// TwinCAT 3 PLC project CAP_TESTER
// ProgramVersion: 3.1.4023.0
// libraries:
//   Tc2_ControllerToolbox, * (Beckhoff Automation GmbH)
//   Tc2_Standard, * (Beckhoff Automation GmbH)
//   Tc2_System, * (Beckhoff Automation GmbH)
//   Tc2_Utilities, * (Beckhoff Automation GmbH)
//   Tc3_Module, * (Beckhoff Automation GmbH)
// project tree:
//   DUTs/ BIT2.TcDUT, ST_AnalogCHSelection.TcDUT
//   GVLs/ GVL.TcGVL, HMI_DB.TcGVL, LV.TcGVL, VoltMonitor_DB.TcGVL
//   / PlcTask.TcTTO
//   POUs/ ADC_10V.TcPOU, ADC_5V.TcPOU, ALIAS.TcPOU, ANALOGConversion.TcPOU, Automated_Capacitor_Test_ST.TcPOU, CounterUP.TcPOU, handleFAULT.TcPOU, handlesensorlimitFAULTS.TcPOU, handlesoftEXCEPTION.TcPOU, HMI.TcPOU, LV_ALIAS.TcPOU, MAIN.TcPOU, Norm_x.TcPOU, PRG_FB_CTRL_PWM_OUT.TcPOU, VoltMonitor.TcPOU
//   POUs/Functions/AnalogIN-ScaleOffset/ AI2temp.TcPOU, AI1temp.TcPOU, AI3temp.TcPOU, AI4temp.TcPOU
//   POUs/Functions/AnalogIN-ScaleOffset/Voltage Calibration/ AI5volt.TcPOU
//   POUs/Functions/AnalogOut-ScaleOffset/ volt_TO_AO1_802L50kV.TcPOU
//   POUs/Functions/ estimatedchargeTIME_802L.TcPOU, HV_Monitor.TcPOU, instantexpectedcapVOLT_802L.TcPOU, Heartbeat.TcPOU, Norm_x_UINT.TcPOU, tempSAFE.TcPOU
// real-time tasks:
//   TASK PlcTask: cycle T#10ms, priority 20, ADS port 350
// I/O:
//   DEVICE Device 1 (EtherCAT), AmsNetId 172.25.226.104.2.1
//     Term 1 (EK1200) [EK1200-5000 EtherCAT Power supply (2A E-Bus)]
//       Term 2 (EL1008) [EL1008 8Ch. Dig. Input 24V, 3ms]
//       Term 3 (EL1008) [EL1008 8Ch. Dig. Input 24V, 3ms]
//       Term 4 (EL2008) [EL2008 8Ch. Dig. Output 24V, 0.5A]
//       Term 5 (EL2008) [EL2008 8Ch. Dig. Output 24V, 0.5A]
//       Term 6 (EL3064) [EL3064 4Ch. Ana. Input 0-10V]
//       Term 7 (EL3064) [EL3064 4Ch. Ana. Input 0-10V]
//       Term 8 (EL3064) [EL3064 4Ch. Ana. Input 0-10V]
//       Term 9 (EL4132) [EL4132 2Ch. Ana. Output +/-10V, 16bit]
//       Term 10 (EL9011) [EL9011 End Terminal]
//   DEVICE Device 3 (RT-Ethernet Protocol) (disabled), AmsNetId 172.25.226.104.4.1
//   DEVICE Device 2 (NOV-DP-RAM) (disabled)
//   DEVICE Device 6 (EtherCAT), AmsNetId 5.97.49.116.7.1
//     Box 11 (170357) [170357]
// variable links:
//   CAP_TESTER/CAP_TESTER Instance <-> Device 1 (EtherCAT)/Term 1 (EK1200)/Term 2 (EL1008)
//     PlcTask Inputs/GVL.PLC_DI{1..8} <-> Channel {1..8}/Input  (8 links)
//   CAP_TESTER/CAP_TESTER Instance <-> Device 1 (EtherCAT)/Term 1 (EK1200)/Term 3 (EL1008)
//     PlcTask Inputs/GVL.PLC_DI{9..16} <-> Channel {1..8}/Input  (8 links)
//   CAP_TESTER/CAP_TESTER Instance <-> Device 1 (EtherCAT)/Term 1 (EK1200)/Term 4 (EL2008)
//     PlcTask Outputs/GVL.PLC_DO{1..8} <-> Channel {1..8}/Output  (8 links)
//   CAP_TESTER/CAP_TESTER Instance <-> Device 1 (EtherCAT)/Term 1 (EK1200)/Term 5 (EL2008)
//     PlcTask Outputs/GVL.PLC_DO{9..16} <-> Channel {1..8}/Output  (8 links)
//   CAP_TESTER/CAP_TESTER Instance <-> Device 1 (EtherCAT)/Term 1 (EK1200)/Term 6 (EL3064)
//     PlcTask Inputs/GVL.PLC_AI{1..4} <-> AI Standard Channel {1..4}/Value  (4 links)
//     PlcTask Inputs/GVL.PLC_AI{1..4}_LIM1 <-> AI Standard Channel {1..4}/Status  (4 links)
//   CAP_TESTER/CAP_TESTER Instance <-> Device 1 (EtherCAT)/Term 1 (EK1200)/Term 7 (EL3064)
//     PlcTask Inputs/GVL.PLC_AI{5..8} <-> AI Standard Channel {1..4}/Value  (4 links)
//     PlcTask Inputs/GVL.PLC_AI{5..8}_LIM1 <-> AI Standard Channel {1..4}/Status  (4 links)
//   CAP_TESTER/CAP_TESTER Instance <-> Device 1 (EtherCAT)/Term 1 (EK1200)/Term 8 (EL3064)
//     PlcTask Inputs/GVL.PLC_AI{9..12} <-> AI Standard Channel {1..4}/Value  (4 links)
//     PlcTask Inputs/GVL.PLC_AI{9..12}_LIM1 <-> AI Standard Channel {1..4}/Status  (4 links)
//   CAP_TESTER/CAP_TESTER Instance <-> Device 1 (EtherCAT)/Term 1 (EK1200)/Term 9 (EL4132)
//     PlcTask Outputs/GVL.PLC_AO1 <-> Channel 1/Output
//     PlcTask Outputs/GVL.PLC_AO2 <-> Channel 2/Output
//   CAP_TESTER/CAP_TESTER Instance <-> Device 6 (EtherCAT)/Box 11 (170357)
//     PlcTask Inputs/GVL.B170357_CapRaw[{0..24}] <-> HV Cap process data mapping/Cap {0..24} Raw  (25 links)

CONFIGURATION CAP_TESTER
    RESOURCE PLC ON TwinCAT3
        TASK PlcTask(INTERVAL := T#10ms, PRIORITY := 20);
        PROGRAM MAIN WITH PlcTask : MAIN;
    END_RESOURCE
END_CONFIGURATION

// ---- DUTs/BIT2.TcDUT
(* STRUCT typedef for EL3XXX AI BIT2 limit *)
TYPE BIT2 :
STRUCT
	BIT_0: BIT;		// < or =< is BIT0 true 
	BIT_1: BIT;		// > or => is BIT1 true
END_STRUCT
END_TYPE

// ---- DUTs/ST_AnalogCHSelection.TcDUT
TYPE ST_AnalogCHSelection :
STRUCT
	b0 : BIT;
	b1 : BIT;
	b2 : BIT;
	b3 : BIT;
END_STRUCT
END_TYPE

// ---- GVLs/GVL.TcGVL
{attribute 'qualified_only'}
VAR_GLOBAL

 //Alwas True & False
 AlwaysTrue : BOOL := TRUE;
 AlwaysFalse : BOOL := FALSE;
 
(* PLC Physical IO *)
	// Digital IO
	buttonSTOP : BOOL;		// Unused
	mechINTERLOCK : BOOL;
	softdump : BOOL := FALSE; 
	softdump_contact : BOOL;   // soft dump relay feedback. Normally Closed - ctrl box dump feedback is the soft dump feedback, in here ctrlbox dump feedback is not used
	chargeCOIL : BOOL := FALSE;
	chargeCOIL_contact : BOOL; // charge coil relay feedback. Normally Open
	shotCOIL : BOOL := FALSE;
	shotCOILrdy : BOOL;
	testFAULTlight : BOOL;
	testRUNlight : BOOL;
	scopetrigger : BOOL;
	charging_alarm :BOOL;
	sparkdetect :BOOL;
	FireDetected :BOOL;  //Newly added for Fire Detection Test
	chrg_to_fire_trig :BOOL := FALSE; //debug signal for Firedetect system
	FruitStandDumpingON : BOOL := FALSE;
	
	(* For HVPS Controller IO *)
	psuVmonitor : INT;		// PLC in to V monitor, is psu V measurement. AI
	psuVCTRL : INT;		// PLC out to remote voltage, is psu V control. AO
	selectREMOTE : BOOL := FALSE;		// PLC out to remote/ local select, is psu ON/ OFF control.
	psuInhibit : BOOL := TRUE;		// PLC out to inhibit, inhibits psu.
	psuInhibit_contact : BOOL;		// No PCB with available signal thus unused.
	psuONOFF : BOOL;		// PLC in to High Voltage Monitor, is psu ON/ OFF status.
	EOCstatus : BOOL;		// PLC in to EOC, is psu End of Charge
	psuINTERLOCK : BOOL;		// PLC in
	psusumFAULT : BOOL;		// PLC in
	psuMaxOutput : UINT;  //Maximum output setting on a Charger Power supply  (12kV or 50kV) * added oct 12, 2022 GL
	
	sparkCharger_ON : BOOL;  // added output to turn on spark charger sept 21, 2022 GL
	sparkCharger_SP_Enable : BOOL; // added setpoint enable to spark charger sept 21, 2022 GL
	
	(* AI TEMP/ VOLT *)
	rawTEMPcap1 : INT; // Cap1 
		TEMPcap1 : INT;
	rawTEMPdump : INT; // Soft Dump
		TEMPdump : INT;
	rawTEMPload : INT; // Load 
		TEMPload : INT;
	rawTEMPambient : INT; // Ambient 
		TEMPambient : INT;
	rawVcap1 : INT;	// Cap1 Voltage
		Vcap1 : INT;
		changeAI5 :BOOL := FALSE;
	raw_HV_monitor : INT;
		HV_monitor :INT;
		
		Vcap2 : INT;  //Cap1 Voltage with 0-10V for testing oct, 27, 2022
		Vcap2_norm : REAL;
		Vcap2_REAL : REAL;
		
	raw_Spark_gap_voltage :INT;  //AI8 - added Oct 5, 2022 - GL
		Spark_gap_voltage :INT;
		Spark_gap_voltage_norm : REAL;
		Spark_gap_voltage_REAL : REAL;
	raw_VoltageMonitor : INT;
(* PLC Internal *)
	appRUN : BOOL;
	

	(* Manual HMI Controls *)
	HMIhold : BOOL;
	HMIcharge : BOOL;
	HMIdump : BOOL;
	HMIshoot : BOOL;
	HMIready : BOOL;
	
(* FAULTS *)
	chargeFAULT : BOOL := FALSE;
	dischargeFAULT : BOOL := FALSE;
	holdFAULT : BOOL := FALSE;
	cap1tempFAULT : BOOL := FALSE;
	ambienttempFAULT : BOOL := FALSE;
	loadtempFAULT : BOOL := FALSE;  // ADDED OCT 14, 2022 GL
	psuFAULT : BOOL := FALSE;
	ctrlsysFAULT : BOOL := FALSE;		// Relates to FB sys
		softdumpFB_FAULT : BOOL := FALSE;
		chargeFB_FAULT : BOOL := FALSE;
		HVpsuFB_FAULT : BOOL := FALSE;
	softexceptionFAULT : BOOL := FALSE;
	test_interval_fault : BOOL := FALSE;
	PreFire_Fault : BOOL := FALSE;

(*DEBUG*)
	ctrl_box_charge_feedback : BOOL;  //relay contact ??
	ctrl_box_dump_feedback : BOOL;	//relay contact ??
(* Start PLC ALIAS *)
		// Digital In
	PLC_DI1 AT %I* : BOOL;
	PLC_DI2 AT %I* : BOOL;
	PLC_DI3 AT %I* : BOOL;
	PLC_DI4 AT %I* : BOOL;
	PLC_DI5 AT %I* : BOOL;
	PLC_DI6 AT %I* : BOOL;
	PLC_DI7 AT %I* : BOOL;
	PLC_DI8 AT %I* : BOOL;
	PLC_DI9 AT %I* : BOOL;
	PLC_DI10 AT %I* : BOOL;
	PLC_DI11 AT %I* : BOOL;
	PLC_DI12 AT %I* : BOOL;
	PLC_DI13 AT %I* : BOOL;
	PLC_DI14 AT %I* : BOOL;
	PLC_DI15 AT %I* : BOOL;
	PLC_DI16 AT %I* : BOOL;
		// Digital Out
	PLC_DO1 AT %Q* : BOOL;
	PLC_DO2 AT %Q* : BOOL;
	PLC_DO3 AT %Q* : BOOL;
	PLC_DO4 AT %Q* : BOOL;
	PLC_DO5 AT %Q* : BOOL;
	PLC_DO6 AT %Q* : BOOL;
	PLC_DO7 AT %Q* : BOOL;
	PLC_DO8 AT %Q* : BOOL;
	PLC_DO9 AT %Q* : BOOL;
	PLC_DO10 AT %Q* : BOOL;
	PLC_DO11 AT %Q* : BOOL;
	PLC_DO12 AT %Q* : BOOL; //Voltage Monitor b0
	PLC_DO13 AT %Q* : BOOL; //Voltage Monitor b1
	PLC_DO14 AT %Q* : BOOL; //Voltage Monitor b2
	PLC_DO15 AT %Q* : BOOL; //Voltage Monitor b3
	PLC_DO16 AT %Q* : BOOL; //spare
		// Analog In
	PLC_AI1 AT %I* : INT;
	PLC_AI2 AT %I* : INT;
	PLC_AI3 AT %I* : INT;
	PLC_AI4 AT %I* : INT;
	PLC_AI5 AT %I* : INT;
	PLC_AI6 AT %I* : INT;
	PLC_AI7 AT %I* : INT;
	PLC_AI8 AT %I* : INT;
	PLC_AI9 AT %I* : INT;
	PLC_AI10 AT %I* : INT;
	PLC_AI11 AT %I* : INT;
	PLC_AI12 AT %I* : INT;
			// Analog Satus Limit WORD Bits 2/3 is Limit 1..... BIT.0 is WORD.2 and BIT.1 is WORD.3
			PLC_AI1_LIM1 AT %I*: WORD;
			PLC_AI2_LIM1 AT %I*: WORD;
			PLC_AI3_LIM1 AT %I*: WORD;
			PLC_AI4_LIM1 AT %I*: WORD;
			PLC_AI5_LIM1 AT %I*: WORD;
			PLC_AI6_LIM1 AT %I*: WORD;
			PLC_AI7_LIM1 AT %I*: WORD;
			PLC_AI8_LIM1 AT %I*: WORD;
			PLC_AI9_LIM1 AT %I*: WORD;
			PLC_AI10_LIM1 AT %I*: WORD;
			PLC_AI11_LIM1 AT %I*: WORD;
			PLC_AI12_LIM1 AT %I*: WORD;
		// Analog Out
	PLC_AO1 AT %Q* : INT;
	PLC_AO2 AT %Q* : INT;
	
	// PLC IO Status
	PLC_EL1008_1 AT %I* : UINT;
	PLC_EL1008_2 AT %I* : UINT;
	PLC_EL2008_1 AT %I* : UINT;
	PLC_EL2008_2 AT %I* : UINT;
	PLC_EL3064_1 AT %I* : UINT;
	PLC_EL3064_2 AT %I* : UINT;
	PLC_EL3064_3 AT %I* : UINT;
	PLC_EL4132_1 AT %I* : UINT;
	
	// EtherCAT Module
	DevCtrl AT %Q* : UINT;
	
	//customed board 170357
	(*B170357_CapRaw0 AT %I* : UINT;
	B170357_CapRaw1 AT %I* : UINT;
	B170357_CapRaw2 AT %I* : UINT;
	B170357_CapRaw3 AT %I* : UINT;
	B170357_CapRaw4 AT %I* : UINT;
	B170357_CapRaw5 AT %I* : UINT;
	B170357_CapRaw6 AT %I* : UINT;
	B170357_CapRaw7 AT %I* : UINT;
	B170357_CapRaw8 AT %I* : UINT;
	B170357_CapRaw9 AT %I* : UINT;
	B170357_CapRaw10 AT %I* : UINT;
	B170357_CapRaw11 AT %I* : UINT;
	B170357_CapRaw12 AT %I* : UINT;
	B170357_CapRaw13 AT %I* : UINT;
	B170357_CapRaw14 AT %I* : UINT;
	B170357_CapRaw15 AT %I* : UINT;
	B170357_CapRaw16 AT %I* : UINT;
	B170357_CapRaw17 AT %I* : UINT;
	B170357_CapRaw18 AT %I* : UINT;
	B170357_CapRaw19 AT %I* : UINT;
	B170357_CapRaw20 AT %I* : UINT;
	B170357_CapRaw21 AT %I* : UINT;
	B170357_CapRaw22 AT %I* : UINT;
	B170357_CapRaw23 AT %I* : UINT;
	B170357_CapRaw24 AT %I* : UINT;*)
	
	B170357_CapRaw AT %I* : ARRAY[0..24] OF UINT;
	B170357_BatLevel AT %I* : BOOL;
	B170357_Heartbeat AT %I* : BOOL;
	

END_VAR

VAR_GLOBAL PERSISTENT
	(* HMI IO *)
	hmiSTOP : BOOL; // In (Into PLC from LabView)
	hmiSTART : BOOL;	// In
	HOA : BOOL;	// In
	
	voltage_held_by_PSU :BOOL;
	isnotSCRhvswitch : BOOL;	// If HV switch has feedback. SCR has ready feedback signal.
	psu50kV_OutputSelected : BOOL; 
	Cap_ratedVoltage : UINT; // unit is in V
	targetVolt_exceed_CapRating_FAULT : BOOL;
	expectedvoltage : INT;
	psuTargetinvolt_echo : DINT;
	
	clearFAULT : BOOL;	// In
	
	testintervalsecs : INT; 	// In
	overall_cycle_time : INT;
	circuitcapacitanceuF : REAL;	// In
	cap1THRESHOLDcel : INT;	// In
	softdumpTHRESHOLDcel : INT := 95; // IN, added oct 14, 2022 GL
	loadTHRESHOLDcel : INT := 95;  // IN, added oct 14, 2022 GL
	ambientTHRESHOLDcel : INT := 95;  // IN, added oct 14, 2022 GL
	allTemperatureInRange : BOOL; //OUT, added oct 14, 2022 GL
	
	targetPSUVOLT : DINT;	// In 
	psuVOLTrating : DINT;	// In
	psuPOWERpeak : DINT;	// In
	chargeTIME : REAL;	// Out. Is estimated charge time of cap
	chargeTIMEmanual : REAL;	// In
	holdTIMEsec : REAL; // IN 
		holdTIMEtime : TIME;
	testNUM: INT;
	testNUMmax : INT;	// In
	testNUMexceed: BOOL;  //CHANGED FROM INT TO BOOL - JUNE 20, 2022
	resettestNUM : BOOL;	// In
	
	(* Current Control *)
	control_current : BOOL;
	duty_cycle : REAL;
	
	InstrumentationFault : BOOL := FALSE;
	noFaultDetected: BOOL := TRUE;
END_VAR

// ---- GVLs/HMI_DB.TcGVL
{attribute 'qualified_only'}
VAR_GLOBAL
	Fault: WORD; 
	
	Charging			: BOOL := FALSE;
	Dumping				: BOOL := FALSE;
	ActivateChargePB 	: BOOL := FALSE;
	ActivateDumpPB 		: BOOL := FALSE;
	
END_VAR

// ---- GVLs/LV.TcGVL
{attribute 'qualified_only'}
// variables to be used with LabVIEW
VAR_GLOBAL
	
aBools : ARRAY[1..20] OF BOOL;
aInts : ARRAY[1..10] OF INT;

END_VAR

// ---- GVLs/VoltMonitor_DB.TcGVL
{attribute 'qualified_only'}
VAR_GLOBAL
	Heartbeat : BOOL;
	BateryOn  : BOOL;
	Channel	: USINT; //ST_AnalogCHSelection;
	VoltageReading_raw : ARRAY[0..24] OF INT;
	VoltageReading_norm : ARRAY[0..24] OF REAL;
	VoltageReading	: ARRAY[0..15] OF REAL;
	LoadMaxRatedV	: REAL := 13800; //-2k TO 35kV
	LoadMinRatedV	: REAL := -1450; //Jake's lab result
	
	CapRaw : ARRAY[0..24] OF UINT;
	CapRawBIT : UINT;
	CapRaw_DummySnap : ARRAY[0..24] OF UINT;
	CapRaw_Str: STRING;
	BatteryLevel : BOOL;
	
	//cunter for missing packets
	missedCTU : CTU;
	//ONS	: R_TRIG;
	missingCNT : WORD :=0;
	
	Time1		: TON;
	Time1_ET	: TIME;
	packetsPerMin : REAL;
	//missedCTU : CTU;
	ONS	: R_TRIG;
	//missingCNT : WORD;
	missingCNT_REAL : REAL;
END_VAR

// ---- POUs/MAIN.TcPOU
PROGRAM MAIN

ALIAS();
LV_ALIAS();
ANALOGconversion();
handleFAULT();
handlesensorlimitFAULTS();
handlesoftEXCEPTION();
Automated_Capacitor_Test_ST();	
HMI();
HV_Monitor();
VoltMonitor();
//HMI Refresh clock
Heartbeat();
// runningLIGHTS();

END_PROGRAM

// ---- POUs/ALIAS.TcPOU
PROGRAM ALIAS
VAR
END_VAR

(* ALIAS Map 
Can be used for wiring and variable linking. ! Remember to SETUP and link AI1-4 LIMIT1 Bits !
Disclaimers: 
Digital IO PCB input Ch3/4 are inverted - No light in, 24V. Wired to PLC_DO6/7
Look at specifcations document for mapping.
*)
	// Digital Input
	GVL.mechINTERLOCK 			:= GVL.PLC_DI1 ;	// Normally Low when not interlock
	GVL.softdump_contact 		:= GVL.PLC_DI2 ;		// NL when no FB. Goes high when the relay is engaged and is not soft dumping. NO 
	GVL.psuONOFF 				:= GVL.PLC_DI3 ;	// To PSU High Voltage Monitor - Normally HIGH when HV OFF/ sig
	GVL.psusumFAULT 			:= GVL.PLC_DI4 ;	// To PSU Sum Fault - NH when no fault/ sig
	//GVL.psuINTERLOCK 			:= GVL.PLC_DI5 ;	// To PSU Interlock. Unknown if NH or NL
	GVL.ctrl_box_dump_feedback 	:= GVL.PLC_DI5;		// this variable is not used, softdump_contact is used instead and it is coming from the ctrlbox dump fb
	GVL.EOCStatus 				:= GVL.PLC_DI6 ;		// End of charge - NH when not EOC
	GVL.sparkdetect 			:= GVL.PLC_DI7 ;		// DI Extra1 - Mech TEST STOP sw - Normally LOW. Not used.
	GVL.chargeCOIL_contact 		:= GVL.PLC_DI8 ;	// NL
	GVL.shotCOILrdy 			:= GVL.PLC_DI9 ;		// NL
	GVL.FireDetected 			:= GVL.PLC_DI10 ;   // for Fire Detection
	GVL.FruitStandDumpingON		:= GVL.PLC_DI13;
	VoltMonitor_DB.Heartbeat 	:= GVL.B170357_Heartbeat;//:= GVL.PLC_DI11 ;   // Voltage Monitor Heartbeat
	VoltMonitor_DB.BateryOn		:= GVL.B170357_BatLevel;//:= GVL.PLC_DI12 ;
	VoltMonitor_DB.CapRaw[0]	:= GVL.B170357_CapRaw[0];
	VoltMonitor_DB.CapRaw[1]	:= GVL.B170357_CapRaw[1];
	VoltMonitor_DB.CapRaw[2]	:= GVL.B170357_CapRaw[2];
	VoltMonitor_DB.CapRaw[3]	:= GVL.B170357_CapRaw[3];
	VoltMonitor_DB.CapRaw[4]	:= GVL.B170357_CapRaw[4];
	VoltMonitor_DB.CapRaw[5]	:= GVL.B170357_CapRaw[5];
	VoltMonitor_DB.CapRaw[6]	:= GVL.B170357_CapRaw[6];
	VoltMonitor_DB.CapRaw[7]	:= GVL.B170357_CapRaw[7];
	VoltMonitor_DB.CapRaw[8]	:= GVL.B170357_CapRaw[8];
	VoltMonitor_DB.CapRaw[9]	:= GVL.B170357_CapRaw[9];
	VoltMonitor_DB.CapRaw[10]	:= GVL.B170357_CapRaw[10];
	VoltMonitor_DB.CapRaw[11]	:= GVL.B170357_CapRaw[11];
	VoltMonitor_DB.CapRaw[12]	:= GVL.B170357_CapRaw[12];
	VoltMonitor_DB.CapRaw[13]	:= GVL.B170357_CapRaw[13];
	VoltMonitor_DB.CapRaw[14]	:= GVL.B170357_CapRaw[14];
	VoltMonitor_DB.CapRaw[15]	:= GVL.B170357_CapRaw[15];
	VoltMonitor_DB.CapRaw[16]	:= GVL.B170357_CapRaw[16];
	VoltMonitor_DB.CapRaw[17]	:= GVL.B170357_CapRaw[17];
	VoltMonitor_DB.CapRaw[18]	:= GVL.B170357_CapRaw[18];
	VoltMonitor_DB.CapRaw[19]	:= GVL.B170357_CapRaw[19];
	VoltMonitor_DB.CapRaw[20]	:= GVL.B170357_CapRaw[20];
	VoltMonitor_DB.CapRaw[21]	:= GVL.B170357_CapRaw[21];
	VoltMonitor_DB.CapRaw[22]	:= GVL.B170357_CapRaw[22];
	VoltMonitor_DB.CapRaw[23]	:= GVL.B170357_CapRaw[23];
	VoltMonitor_DB.CapRaw[24]	:= GVL.B170357_CapRaw[24];
	(*GVL. := GVL.PLC_DI13 ;
	GVL. := GVL.PLC_DI14 ;
	GVL. := GVL.PLC_DI15 ;
	GVL. := GVL.PLC_DI16 ;
	*)
	
		// Digital Out
	GVL.PLC_DO1 := GVL.shotCOIL ;	// NO
	GVL.PLC_DO2 := GVL.softdump ;	// NC
	GVL.PLC_DO3 := GVL.psuInhibit ;	// To PSU Inhibit - NO
	GVL.PLC_DO4 := GVL.selectREMOTE ;		// To PSU Remote/ Local Select - NO
	GVL.PLC_DO5 := GVL.chargeCOIL ;		// To charge SSR - NO
	GVL.PLC_DO6 := GVL.scopetrigger ;	// NO - To scope trigger
		
	GVL.PLC_DO7 := GVL.testNUMexceed ;
	GVL.PLC_DO8 := GVL.charging_alarm ;
	GVL.PLC_DO9 := GVL.chrg_to_fire_trig ;   
	GVL.PLC_DO10 := GVL.sparkCharger_ON;  // added for the spark charger power supply sept 21, 2022 GL
	GVL.PLC_DO11 := GVL.sparkCharger_SP_Enable; // added for the spark charger power supply sept 21, 2022 GL
	GVL.PLC_DO12 := VoltMonitor_DB.Channel.0; //a0
	GVL.PLC_DO13 := VoltMonitor_DB.Channel.1; //a1
	GVL.PLC_DO14 := VoltMonitor_DB.Channel.2;
	GVL.PLC_DO15 := VoltMonitor_DB.Channel.3;
	(*GVL.PLC_DO16 := GVL. ;
	*)
	
		// Analog In
			// AI1-4 has 4mA lower limit fault bits *)
	GVL.rawTEMPcap1 := GVL.PLC_AI1 ;
	GVL.rawTEMPdump := GVL.PLC_AI2 ;
	GVL.rawTEMPload := GVL.PLC_AI3 ;
	GVL.rawTEMPambient := GVL.PLC_AI4 ;
	GVL.rawVcap1 := GVL.PLC_AI5 ;
	GVL.psuVmonitor := GVL.PLC_AI6 ;	// To PSU V Monitor. Not used
	GVL.raw_HV_monitor := GVL.PLC_AI7  ;
	
	GVL.raw_Spark_gap_voltage := GVL.PLC_AI8 ;
	GVL.raw_VoltageMonitor := GVL.PLC_AI9 ;
	(*GVL. := GVL.PLC_AI10 ;
	GVL. := GVL.PLC_AI11 ;
	GVL. := GVL.PLC_AI12 ;
	*)
		// Analog In - LIMITs (These are directly linked, check GVLs)
		
		// Analog Out
	GVL.PLC_AO1 := GVL.psuVCTRL ;	// To PSU Remote Voltage
	(*
	GVL.PLC_AO2 := GVL. ;
	*)
	
	// Ethernet (These are directly linked)

END_PROGRAM

// ---- POUs/Functions/Heartbeat.TcPOU
PROGRAM Heartbeat
VAR
	start_TON: TON;
	start_TON_et : TIME;
	reset_TON : TON;
	reset_TON_et : TIME;
	screen_refresh_pulse : BOOL;
	
	pulse_ms_TON : TON;
	pulse_ms_et : TIME;
	reset_ms_TON : TON;
	reset_ms_TON_et : TIME;
	pulse_ms : BOOL;
END_VAR

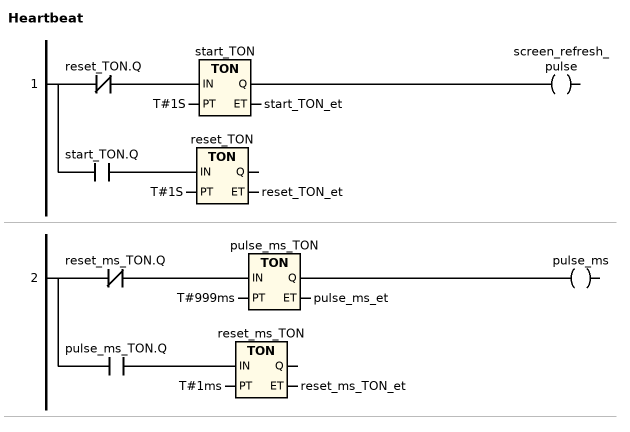
// NETWORK 1
start_TON(IN := NOT reset_TON.Q, PT := T#1S, ET => start_TON_et); // TON
screen_refresh_pulse := start_TON.Q;
reset_TON(IN := start_TON.Q, PT := T#1S, ET => reset_TON_et); // TON

// NETWORK 2
pulse_ms_TON(IN := NOT reset_ms_TON.Q, PT := T#999ms, ET => pulse_ms_et); // TON
pulse_ms := pulse_ms_TON.Q;
reset_ms_TON(IN := pulse_ms_TON.Q, PT := T#1ms, ET => reset_ms_TON_et); // TON

END_PROGRAM

// ---- POUs/LV_ALIAS.TcPOU
PROGRAM LV_ALIAS
VAR
END_VAR

// sole purpose of this PRG is to build arrays that LabVIEW can easily read
LV.aBools[1] := GVL.chargeFAULT;
LV.aBools[2] := GVL.dischargeFAULT;
LV.aBools[3] := GVL.holdFAULT;
LV.aBools[4] := GVL.cap1tempFAULT;
LV.aBools[5] := GVL.ambienttempFAULT;
LV.aBools[6] := GVL.psuFAULT;
LV.aBools[7] := GVL.ctrlsysFAULT;
LV.aBools[8] := GVL.appRUN;
LV.aBools[9] := GVL.softdumpFB_FAULT;
LV.aBools[10] := GVL.chargeFB_FAULT;
LV.aBools[11] := GVL.HVpsuFB_FAULT;
LV.aBools[12] := GVL.softexceptionFAULT;
LV.aBools[13] := GVL.EOCstatus;
LV.aBools[14] := GVL.shotCOILrdy;
LV.aBools[15] := GVL.testNUMexceed;
LV.aBools[16] := GVL.scopetrigger;
LV.aBools[17] := GVL.test_interval_fault;
LV.aBools[18] := GVL.targetVolt_exceed_CapRating_FAULT;
LV.aBools[19] := GVL.allTemperatureInRange;
LV.aBools[20] := GVL.loadtempFAULT;

LV.aInts[1] := GVL.testNUM;
LV.aInts[2] := GVL.Vcap1;
LV.aInts[3] := GVL.TEMPcap1;
LV.aInts[4] := GVL.psuVmonitor;
LV.aInts[5] := GVL.TEMPload;
LV.aInts[6] := GVL.TEMPdump;
LV.aInts[7] := GVL.TEMPambient;
LV.aInts[8] := GVL.expectedvoltage;
LV.aInts[9] := GVL.testintervalsecs;
LV.aInts[10] := GVL.Spark_gap_voltage;

END_PROGRAM

// ---- POUs/ANALOGConversion.TcPOU
PROGRAM ANALOGConversion
VAR
	
END_VAR

(* Program converts raw AI values to Cel temperatures or Volts *)
GVL.TEMPcap1 := AI1temp(AI1raw:= GVL.rawTEMPcap1);
GVL.TEMPdump := AI2temp(AI2raw:= GVL.rawTEMPdump);
GVL.TEMPload := AI3temp(AI3raw:= GVL.rawTEMPload);
GVL.TEMPambient := AI4temp(AI4raw:= GVL.rawTEMPambient);
GVL.Vcap1 := AI5volt(AI5voltageraw:= GVL.rawVcap1, isGreaterthanlimit:= GVL.changeAI5);

//GVL.Spark_gap_voltage :=AI5Volt(AI5voltageraw := GVL.raw_Spark_gap_voltage, isGreaterthanlimit:= GVL.changeAI5); 
GVL.Spark_gap_voltage_norm := Norm_x (raw_input := INT_TO_REAL (GVL.raw_Spark_gap_voltage),
										x_max := 32767,
										x_min := 346); //min reading is 346 - this might change depending on the setup.  oct 17, 2022
GVL.Spark_gap_voltage_REAL := 50 * ADC_10V (normal_input := GVL.Spark_gap_voltage_norm, //units is in kV, ie 50kV
									x_max := 10,
									x_min := 0);
GVL.Spark_gap_voltage := REAL_TO_INT (GVL.Spark_gap_voltage_REAL);	// convert it back to INT for ADS Labview oct 06, 2022


//Added vcap2 to see if the current setup is good for 0-10V voltage feedback to opto
GVL.Vcap2_norm := Norm_x (raw_input:= INT_TO_REAL (GVL.rawVcap1),
							x_max := 16384,
							x_min := 1734);
							
GVL.Vcap2_REAL := 40000 * ADC_10V (normal_input := GVL.Vcap2_norm,
								x_max := 10,
								x_min := 0);
								
GVL.Vcap2 := REAL_TO_INT (GVL.Vcap2_REAL);


//adding voltage monitor
(*
VoltMonitor_DB.VoltageReading_norm[0] := Norm_x ( raw_input := INT_TO_REAL(VoltMonitor_DB.VoltageReading_raw[0]),
													x_max := 32767,
													x_min := 2956);
VoltMonitor_DB.VoltageReading[0] := (VoltMonitor_DB.LoadMaxRatedV - VoltMonitor_DB.LoadMinRatedV) * ADC_10V (normal_input := VoltMonitor_DB.VoltageReading_norm[0],
															x_max := 9.8274,
															x_min := 0.0080297);
	*)														
//new voltage monitor board 170357
VoltMonitor_DB.VoltageReading_norm[0] := Norm_x ( raw_input := INT_TO_REAL(VoltMonitor_DB.VoltageReading_raw[0]),
													x_max := 1023,
													x_min := 0);
VoltMonitor_DB.VoltageReading[0] := (VoltMonitor_DB.LoadMaxRatedV - VoltMonitor_DB.LoadMinRatedV) * VoltMonitor_DB.VoltageReading_norm[0] - 1450;

END_PROGRAM

// ---- POUs/Functions/AnalogIN-ScaleOffset/AI1temp.TcPOU
FUNCTION AI1temp : INT
VAR_INPUT
	AI1raw : INT;
END_VAR
VAR
END_VAR

(* Description: 
Function performs the 0-32767 offset+scaling+interpretation to a Cel temp for AI0. Matched to PWM Reciever board CH1
EL3XXX converts the interpreted 0-32767 value into voltage.
Voltage is converted to temperature using a calibrated formula: (scale*volt)-offset=temp

For IR sensor Ch1*)
AI1temp := REAL_TO_INT( ((1.842963*(INT_TO_REAL(AI1raw)*0.0003049947521145891)+4)-4.0 ) *450.0/16.0 - 70.0 ) ;
// Calibrated Dec 9, 2021.

END_FUNCTION

// ---- POUs/Functions/AnalogIN-ScaleOffset/AI2temp.TcPOU
FUNCTION AI2temp : INT
VAR_INPUT
	AI2raw : INT;
END_VAR
VAR
END_VAR

(* Description: 
Function performs the 0-32767 offset+scaling+interpretation to a Cel temp for AI0. Matched to PWM Reciever board CH2
EL3XXX converts the interpreted 0-32767 value into voltage.
Voltage is converted to temperature using a calibrated formula: (scale*volt)-offset=temp

For IR sensor Ch2*)
AI2temp := REAL_TO_INT( (( INT_TO_REAL(AI2raw)*0.0005206935248569184154 + 3.0517032207384131972)-4.0 ) *450.0/16.0 - 69.0) ;
// Calibrated Dec 9, 2021.

END_FUNCTION

// ---- POUs/Functions/AnalogIN-ScaleOffset/AI3temp.TcPOU
FUNCTION AI3temp : INT
VAR_INPUT
	AI3raw : INT;
END_VAR
VAR
END_VAR

(* Description: 
Function performs the 0-32767 offset+scaling+interpretation to a Cel temp for AI0. Matched to PWM Reciever board CH3
EL3XXX converts the interpreted 0-32767 value into voltage.
Voltage is converted to temperature using a calibrated formula: (scale*volt)-offset=temp

For IR sensor Ch3*)
AI3temp := REAL_TO_INT( ((1.842963*(INT_TO_REAL(AI3raw)*0.0003049947521145891)+4)-4.0 ) *450.0/16.0 - 70.0 ) ;
//AI3temp := REAL_TO_INT( (( INT_TO_REAL(AI3raw)*0.0005058939598786860088 + 3.3586439434355245368)-4.0 ) *450.0/16.0 - 31.0) ;
// Calibrated Dec 9, 2021.

END_FUNCTION

// ---- POUs/Functions/AnalogIN-ScaleOffset/AI4temp.TcPOU
FUNCTION AI4temp : INT
VAR_INPUT
	AI4raw : INT;
END_VAR
VAR
END_VAR

(* Description: 
Function performs the 0-32767 offset+scaling+interpretation to a Cel temp for AI0. Matched to PWM Reciever board CH4
EL3XXX converts the interpreted 0-32767 value into voltage.
Voltage is converted to temperature using a calibrated formula: (scale*volt)-offset=temp

For ambient thermocouple Ch4*)
AI4temp := REAL_TO_INT( ( (0.0005242592739693383113*INT_TO_REAL(AI4raw)) + 2.9817690444038446262) * 30.138875 - 117 ) ;
// Calibrated Dec 9, 2021

END_FUNCTION

// ---- POUs/Functions/AnalogIN-ScaleOffset/Voltage Calibration/AI5volt.TcPOU
FUNCTION AI5volt : INT
VAR_INPUT
	AI5voltageraw : INT;
	isGreaterthanlimit :BOOL;
END_VAR
VAR
	voltageraw : REAL;
END_VAR
VAR_OUTPUT
END_VAR

(* This function performs the 0-32767 offset+scaling+interpretation to a voltage for AI4.
Function specifically FOR 17-0184B-20kV probe, PWM reciever board CH5 *)

// For positive HV probe with R7 para res mod: AI4volt := REAL_TO_INT( (INT_TO_REAL(AI5voltageraw)*(-0.66444986951763616461) ) + 19314.84300025254651 );
// Look at specifications document. Calibrated Dec 8, 2021.
//VM Calibration
voltageraw := INT_TO_REAL(AI5voltageraw);
IF voltageraw >= 4799 THEN
	AI5volt := REAL_TO_INT (0.598211701572909*voltageraw - 908.007762297163000);
ELSE
	AI5volt := REAL_TO_INT (0.646313738227*voltageraw -1101.65962974992);
END_IF

END_FUNCTION

// ---- POUs/Norm_x.TcPOU
FUNCTION Norm_x : REAL
VAR_INPUT
	raw_input : REAL;
	x_max : INT := 32767;
	x_min : INT := 0;
END_VAR
VAR
END_VAR

// 0 - 10V AI INPUT 
Norm_x := (raw_input - x_min) / (x_max - x_min);

END_FUNCTION

// ---- POUs/ADC_10V.TcPOU
FUNCTION ADC_10V : REAL
VAR_INPUT
	normal_input : REAL;
	x_max : REAL := 10;
	x_min : REAL := 0;
END_VAR
VAR
	voltage_reading : REAL;
END_VAR

// 0 - 10V AI INPUT | normal_input 0-100%
voltage_reading := 10 * normal_input;
ADC_10V := (voltage_reading - x_min) / (x_max - x_min);

END_FUNCTION

// ---- POUs/handleFAULT.TcPOU
PROGRAM handleFAULT
VAR
	// Threshold temperatures are hard coded
	// Both defines exist in Automated_Cap_TEST also
	cap1THRESHOLDcel : INT;	
	//ambientTHRESHOLDcel : INT := 40;
	IO_Err : UINT;
	
	R_TRIG1 : R_TRIG;
	F_TRIG1 : F_TRIG;
	genDelay1 : TON;		// General delay - Used to wait for feedback signals
		checkFB1 : BOOL := FALSE;
		iterateDelay1 : BOOL := FALSE;
		elapsedDelay1 : TIME := T#500MS;	
	R_TRIG2 : R_TRIG;
	F_TRIG2 : F_TRIG;
	genDelay2 : TON;		// General delay - Used to wait for feedback signals
		checkFB2 : BOOL := FALSE;
		iterateDelay2 : BOOL := FALSE;
		elapsedDelay2 : TIME := T#500MS;	
	R_TRIG3 : R_TRIG;
	F_TRIG3 : F_TRIG;
	genDelay3 : TON;		// General delay - Used to wait for feedback signals
		checkFB3 : BOOL := FALSE;
		iterateDelay3 : BOOL := FALSE;
		elapsedDelay3 : TIME := T#500MS;
	R_TRIG4 : R_TRIG;
	F_TRIG4 : F_TRIG;	
	genDelay4: TON;		// General delay - Used to wait for feedback signals
		checkFB4 : BOOL := FALSE;
		iterateDelay4 : BOOL := FALSE;
		elapsedDelay4 : TIME := T#500MS;
	(* R_TRIG5 : R_TRIG;
	F_TRIG5 : F_TRIG;
	genDelay5: TOF;		// General delay - Used to wait for feedback signals
		checkFB5 : BOOL := FALSE;
		elapsedDelay5 : TIME;	*)	
		
	FBrtrigQ1 : BOOL;
	FBftrigQ1 : BOOL;
	
	FBrtrigQ2 : BOOL;
	FBftrigQ2 : BOOL;
	
	FBrtrigQ3 : BOOL;
	FBftrigQ3 : BOOL;
	
	FBrtrigQ4 : BOOL;
	FBftrigQ4 : BOOL;
	
	(* FBrtrigQ5 : BOOL;
	FBftrigQ5 : BOOL; *)
	
END_VAR

(* Program deals with capacitor, ambient (Air conditioning fault) temperature faults and fault clears.
Other faults are dealt with within the Automated_Capacitor_Test PGM. *)

//TEMPERATURE FAULTS
// Capacitor and ambient temperature is always monitored and can fault anytime
GVL.TEMPcap1 := AI1temp(AI1raw:= GVL.rawTEMPcap1);
GVL.TEMPambient := AI4temp(AI4raw:= GVL.rawTEMPambient);
IF NOT tempSAFE(TEMPcel:= GVL.TEMPcap1, thresholdTEMPcel:= GVL.cap1THRESHOLDcel) THEN
	GVL.cap1tempFAULT := TRUE;
ELSIF NOT tempSAFE(TEMPcel:= GVL.TEMPambient, thresholdTEMPcel:= GVL.ambientTHRESHOLDcel) THEN
	GVL.ambienttempFAULT := TRUE;
(* For upgrade with 2nd ambient+cap2 temperature sensor for control chamber.
ELSIF NOT tempSAFE(TEMPcel:= GVL.TEMPcap2, thresholdTEMPcel:= GVL.cap1THRESHOLDcel) THEN
	GVL.cap1tempFAULT := TRUE;
ELSIF NOT tempSAFE(TEMPcel:= GVL.TEMPambient2, thresholdTEMPcel:= ambientTHRESHOLDcel) THEN
	GVL.ambienttempFAULT := TRUE;
	*)
END_IF

// LOAD TEMPERATURE FAULT
IF GVL.TEMPload > GVL.loadTHRESHOLDcel THEN
	GVL.loadtempFAULT := TRUE;
	ELSE
		GVL.loadtempFAULT := FALSE;
END_IF;


IF Automated_Capacitor_Test_ST.cap1_Temp = TRUE AND Automated_Capacitor_Test_ST.dump_Temp = TRUE AND Automated_Capacitor_Test_ST.load_Temp = TRUE AND Automated_Capacitor_Test_ST.ambient_Temp = TRUE THEN
	GVL.allTemperatureInRange := TRUE;
	ELSE
		GVL.allTemperatureInRange :=FALSE;
END_IF;

// PSU Fault
IF GVL.psusumFAULT THEN
	GVL.psuFAULT := TRUE;
END_IF

(* FEEDBACK HANDLING with a delay 
The code is built in a way so upon a change event it checks the FB signal after a delay 
Each sys has its own timer. Would have grouped timers but worried about overlap.
Upon a rise/fall edge -> A delay before check. No edge -> no delay check. *)

// Softdump FB
R_TRIG1(CLK:= GVL.softdump, Q=> FBrtrigQ1);
F_TRIG1(CLK:= GVL.softdump, Q=> FBftrigQ1);
IF FBrtrigQ1 OR FBftrigQ1 OR iterateDelay1 THEN		
	iterateDelay1 := TRUE; //First initialization
	elapsedDelay1 := T#0MS;
	genDelay1(IN:= TRUE, PT:= T#500MS, Q=> checkFB1, ET=> elapsedDelay1);
END_IF

IF checkFB1 THEN		// If recently changed variable then use delay, if not recently change just straight to check
	genDelay1(IN:= FALSE, PT:= T#500MS, Q=> checkFB1, ET=> elapsedDelay1);
	elapsedDelay1 := T#0MS;
	iterateDelay1 := FALSE;
	// Start checking FB
	IF (NOT GVL.softdump AND GVL.softdump_contact) OR (GVL.softdump AND NOT GVL.softdump_contact) THEN
		GVL.ctrlsysFAULT := TRUE;
		GVL.softdumpFB_FAULT := TRUE;
	END_IF
END_IF

// Charge Relay FB
R_TRIG2(CLK:= GVL.chargeCOIL, Q=> FBrtrigQ2);
F_TRIG2(CLK:= GVL.chargeCOIL, Q=> FBftrigQ2);
IF FBrtrigQ2 OR FBftrigQ2 OR iterateDelay2 THEN		// Activate for 1 scan
	iterateDelay2 := TRUE;
	elapsedDelay2 := T#0MS;
	genDelay2(IN:= TRUE, PT:= T#500MS, Q=> checkFB2, ET=> elapsedDelay2);
END_IF

IF checkFB2 THEN		// If recently changed variable then use delay, if not recently change just straight to check
	genDelay2(IN:= FALSE, PT:= T#500MS, Q=> checkFB2, ET=> elapsedDelay2);
	elapsedDelay2 := T#00MS;
	iterateDelay2 := FALSE;
	// Start checked systems
	IF (GVL.chargeCOIL AND NOT GVL.chargeCOIL_contact) OR (NOT GVL.chargeCOIL AND GVL.chargeCOIL_contact) THEN
		GVL.ctrlsysFAULT := TRUE;
		GVL.chargeFB_FAULT := TRUE;
	END_IF
END_IF

// PSU HV ON/OFF
R_TRIG3(CLK:= GVL.selectREMOTE, Q=> FBrtrigQ3);
F_TRIG3(CLK:= GVL.selectREMOTE, Q=> FBftrigQ3);
IF FBrtrigQ3 OR FBftrigQ3 OR iterateDelay3 THEN		// Activate for 1 scan
	iterateDelay3 := TRUE;
	elapsedDelay3 := T#0MS;
	genDelay3(IN:= TRUE, PT:= T#500MS, Q=> checkFB3, ET=> elapsedDelay3);
END_IF

IF checkFB3 THEN		// If recently changed variable then use delay, if not recently change just straight to check
	genDelay3(IN:= FALSE, PT:= T#500MS, Q=> checkFB3, ET=> elapsedDelay3);
	elapsedDelay3 := T#00MS;
	iterateDelay3 := FALSE;
	// Start checked systems
	IF (GVL.selectREMOTE AND GVL.psuONOFF) OR (NOT GVL.selectREMOTE AND NOT GVL.psuONOFF) THEN
		GVL.ctrlsysFAULT := TRUE;
		GVL.HVpsuFB_FAULT := TRUE;
	END_IF;
END_IF

(* Removed, 17-0066E has no InhibFB. // PSU Inhibit Feedback
R_TRIG4(CLK:= GVL.psuInhibit, Q=> FBrtrigQ4);
F_TRIG4(CLK:= GVL.psuInhibit, Q=> FBftrigQ4);
IF FBrtrigQ4 OR FBftrigQ4 OR iterateDelay4 THEN		// Activate for 1 scan
	iterateDelay4 := TRUE;
	elapsedDelay4 := T#0MS;
	genDelay4(IN:= TRUE, PT:= T#500MS, Q=> checkFB4, ET=> elapsedDelay4);
END_IF

IF checkFB4 THEN		// If recently changed variable then use delay, if not recently change just straight to check
	genDelay4(IN:= FALSE, PT:= T#500MS, Q=> checkFB4, ET=> elapsedDelay4);
	elapsedDelay4 := T#00MS;
	iterateDelay4 := FALSE;
	// Start checked systems
	IF (GVL.psuInhibit AND GVL.psuInhibitFB) OR (NOT GVL.psuInhibit AND NOT GVL.psuInhibitFB) THEN
		GVL.ctrlsysFAULT := TRUE;
	END_IF;
END_IF *)

//50kV and 12kV powersupply limite selection - oct 14, 2022 GL
IF GVL.psu50kV_OutputSelected = TRUE THEN 
	GVL.psuMaxOutput := 50000;
	ELSE 
		GVL.psuMaxOutput := 12000;
END_IF;

IF GVL.targetPSUVOLT > GVL.Cap_ratedVoltage THEN
	GVL.targetVolt_exceed_CapRating_FAULT := TRUE;
	ELSE
		GVL.targetVolt_exceed_CapRating_FAULT := FALSE;
END_IF;

//Fault Permissives
IF NOT GVL.chargeFAULT AND NOT GVL.dischargeFAULT AND NOT GVL.holdFAULT AND NOT GVL.ctrlsysFAULT AND NOT GVL.cap1tempFAULT AND NOT GVL.ambienttempFAULT
AND NOT GVL.psuFAULT AND NOT GVL.test_interval_fault AND NOT GVL.targetVolt_exceed_CapRating_FAULT THEN //AND GVL.mechINTERLOCK   // psuFAULT, mechinterlock normally high (NH)
	GVL.noFaultDetected := TRUE; //added prefire fault
ELSE
	GVL.noFaultDetected := FALSE;
	END_IF;
IF (GVL.testintervalsecs < 30) THEN
	GVL.test_interval_fault := TRUE;
ELSE
	GVL.test_interval_fault := FALSE;
END_IF

(* Fault clear LOGIC. clearFAULT from LabView *)
IF GVL.clearFAULT AND NOT GVL.appRUN THEN // Momentary PB
	GVL.chargeFAULT := FALSE;
	GVL.dischargeFAULT := FALSE;
	GVL.holdFAULT := FALSE;
	GVL.psuFAULT := FALSE;
	GVL.ctrlsysFAULT := FALSE;
		GVL.softdumpFB_FAULT := FALSE;
		GVL.chargeFB_FAULT := FALSE;
		GVL.HVpsuFB_FAULT := FALSE;
	GVL.cap1tempFAULT := FALSE;
	GVL.ambienttempFAULT := FALSE;
	GVL.softexceptionFAULT := FALSE;
	GVL.loadtempFAULT := FALSE;
	GVL.targetVolt_exceed_CapRating_FAULT := FALSE;
	GVL.PreFire_Fault := FALSE; 
END_IF;


(* PLC Sys FAULTS - In PROGRESS
EL1008 Fault 
IO_Err := 
IF PLC_GVL.PLC_EL1008_1 = 0x001 THEN
END_IF
*)

END_PROGRAM

// ---- POUs/Functions/tempSAFE.TcPOU
FUNCTION tempSAFE : BOOL
VAR_INPUT
	TEMPcel : INT;
	thresholdTEMPcel : INT;
END_VAR
VAR
END_VAR

// If temp passed is under threshold, returns TRUE (is safe)
IF TEMPcel <= thresholdTEMPcel THEN
	tempSAFE := TRUE;
ELSE 
	tempSAFE := FALSE;
END_IF;

END_FUNCTION

// ---- POUs/Automated_Capacitor_Test_ST.TcPOU
PROGRAM Automated_Capacitor_Test_ST
VAR
	// Threshold Temps #DEFINES
	//ambientTHRESHOLDcel : INT := 40; // Exists in handleFAULT pgm also. Change in 2 places
	//loadTHRESHOLDcel : INT := 95;
	//softdumpTHRESHOLDcel : INT := 95;
	
	// #DEFINE
	chrgvoltTOLERANCE 		: INT := 10000;		// Charge Algorithm Voltage Tolerance
	holdvoltThreshold 		: INT := 1000;	// Threshold of allowable decay voltage for cap during hold period
	lowlimtimeTOLERANCE 	: REAL := 1;
	shotrelayDURATION 		: TIME := T#7S;	// Continued activation time of HV shot switch
	firstwaitTIME 			: TIME := T#13S;		// Safety wait timer before test can initiate
	
	// // PLC Status
	processSTEP 			: USINT := 0;
	
		// TIMEs
	estfullchrgTIME 		: REAL;
	chargeTIME 				: REAL;
		chargeTIMEdint 		: DINT;
		chargeTIMEtime 		: TIME;
	beforestartTON 			: TON;
		elapsedbeforestartTIME : TIME;
		startReady 				: BOOL;
	chargeTON 				: TON;
		elapsedChargereal 		: REAL;
		elapsedCharge 			: TIME;
		inhibitVariable 		: BOOL;
	holdTON 				: TON;
		holdTIMEtime 			: TIME;
		elapsedhold 			: TIME;
		shotready 				: BOOL := FALSE;
	holdTON2 				: TON;
		holdTIMEtime2 			: TIME;
		elapsedhold2 			: TIME;
		shotready2 				: BOOL := FALSE;
	shotTON 				: TON;
		shooted 				: BOOL := FALSE;
		elapsedshot 			: TIME;
	testwaitTON 			: TON;
		waitTIMEtime 			: TIME;
		elapsedwait 			: TIME;
		holdtimerQ 				: BOOL;	
	EOCF_TRIG 				: F_TRIG; //End of Charge
		EOCBool 				: BOOL;
	EOCTON 					: TON;
		EOCTIMEtime 			: TIME := T#2000MS;
		elapsedEOC 				: TIME;
		EOCBool2 				: BOOL;
		EOCPassed 				: BOOL;
		iterateEOC 				: BOOL := FALSE;
	extendedChargeTimer 	: TON;
		extendedToleranceTIME 	: TIME := T#15S;
		extendedElapsed 		:TIME;
		extendedTimeReached 	: BOOL;
	Delay 					: TON;
		wait 					: TIME:= T#1S;
		elapsed					: TIME;
		complete				: BOOL := FALSE;
	Delay2 					:TON;
		wait2 					: TIME:= T#1S;
		elapsed2				: TIME;
		complete2				: BOOL := FALSE;
		
	// TEMP Statuses - True means under threshold TEMP
	cap1_Temp 			: BOOL;
	ambient_Temp		: BOOL;
	load_Temp			: BOOL;
	dump_Temp			: BOOL;
	
	// Local Variables
	expectcapVOLT 			: REAL;
	fullCHRG 				: BOOL;
	internalBOOLcharge 		: BOOL := FALSE;
	internalBOOLSDL 		: BOOL := FALSE;
	//Debug Variables
	VoltAtHOLD				: DINT;
	expectedATHOLD			: REAL;
	chrg_time_for_interval 	: TIME;
	// Function Variables - "Static C" variables for iterative functions
	capvoltiter 			: REAL;	
	lasttimesec 			: REAL;
	
	//spark charger
	sparkcharger_TON 		: TON;
	sparkcharger_TON_PT 	: TIME:= T#5S;
	sparkcharger_ready 		: BOOL;
	
	sparkcharger_softdump_TON 	: TON;
	sparkcharger_softdump_PT 	: TIME := T#7S;  //time delay between after shot and soft dump.
	
	hold_betweenCharge_nShot_TON 	: TON;
	hold_betweenCharge_nShot_PT 	: TIME := T#500MS;	
	
	Vcap_sample 					: ARRAY [1..2] OF REAL;
	i 								: INT := 1;
	fbGetSystemTime 				: GETSYSTEMTIME;
	fileTIME 						: T_FILETIME;
	sTIME							: STRING;
END_VAR

// Latching START
IF (GVL.hmiSTART OR GVL.appRUN) AND
(NOT GVL.hmiSTOP // AND NOT GVL.buttonSTOP
AND GVL.noFaultDetected //AND GVL.mechINTERLOCK		// psuFAULT, mechinterlock normally high (NH)
AND NOT GVL.testNUMexceed) THEN
	IF NOT GVL.appRUN THEN		// Handles first run
		processSTEP := 0;
	END_IF;
	GVL.appRUN := TRUE;
	Delay( IN:= FALSE, PT:= wait, Q=>complete, ET=> elapsed);
	complete := FALSE;
	Delay2( IN:= FALSE, PT:= wait2, Q=>complete2, ET=> elapsed2);
	complete2 := FALSE;
// STOP + safe state + landing pad upon fault detection
ELSE 
	GVL.appRUN := FALSE;
	(* Return to safe conditions - Mind order of operation *)
	GVL.shotCOIL := FALSE;
	GVL.psuInhibit := TRUE; 
	Delay( IN:= TRUE, PT:= wait, Q=>complete, ET=> elapsed);
		IF complete THEN
			GVL.chargeCOIL := FALSE;
			GVL.selectREMOTE := FALSE;
			volt_TO_AO1_802L50kV(psuTargetinvolt:= 0, psuMaxOutput:= GVL.psuMaxOutput, VpsuOut:= GVL.psuVCTRL);
			Delay2( IN:= TRUE, PT:= wait2, Q=>complete2, ET=> elapsed2);
				IF complete2 THEN
					GVL.softdump := FALSE; // NC
					Delay( IN:= FALSE, PT:= wait, Q=>complete, ET=> elapsed);
					complete := FALSE;
					Delay2( IN:= FALSE, PT:= wait2, Q=>complete2, ET=> elapsed2);
					complete2 := FALSE;
					elapsed := T#0S;
					elapsed2 := T#0S;
				END_IF;
		END_IF;
	
	// Timer/BOOL/internal logic resets (If test stopped midway. Returns test to default conditions)
	beforestartTON(IN:= FALSE, PT:= T#10S, Q=> startReady, ET=> elapsedbeforestartTIME);
	chargeTON(IN:= FALSE, PT:= chargeTIMEtime, Q=> inhibitVariable, ET=> elapsedCharge );
	holdTON(IN:= FALSE, PT:= holdTIMEtime, Q=> shotready, ET=> elapsedhold);
	shotTON(IN:= FALSE, PT:= T#250MS, Q=> shooted, ET=> elapsedshot);
	testwaitTON(IN:= FALSE, PT:= holdTIMEtime, Q=> holdtimerQ, ET=> elapsedwait);
	
	elapsedbeforestartTIME := T#0MS;
	elapsedCharge := T#0MS;
	internalBOOLcharge := FALSE;
	lasttimesec := 0;
	capvoltiter := 0;
	
	holdTON2(IN:= FALSE, PT:= T#1S, Q=> shotready2, ET=> elapsedhold2);
	shotready2 := FALSE;
	elapsedhold2 := T#0S;
	internalBOOLSDL := FALSE;
	
	EOCPassed := FALSE;
	EOCBool := FALSE;
	EOCBool2 := FALSE;
	EOCTON(IN:= FALSE, PT:= EOCTIMEtime, Q=> EOCBool2, ET=> elapsedEOC);
	
	GVL.charging_alarm := FALSE;
	GVL.chrg_to_fire_trig := FALSE;
	
	extendedChargeTimer(IN :=FALSE, PT:= extendedToleranceTIME,Q => extendedTimeReached, ET =>extendedElapsed);
	extendedElapsed := T#0MS;
	
	elapsedhold := T#0MS;
	elapsedshot := T#0MS;
	elapsedwait := T#0MS;
	
	sparkcharger_TON (IN:= FALSE, PT:= sparkcharger_TON_PT, Q=> sparkcharger_ready);
	sparkcharger_softdump_TON (IN:= FALSE, PT:= sparkcharger_softdump_PT);

	processSTEP := 0;
END_IF;


// Reset Test Number
IF GVL.resettestNUM THEN
	GVL.testNUM := 0;
	GVL.testNUMexceed := FALSE;
END_IF

//calculate cycle time
IF GVL.chargeTIMEmanual <0 THEN
	GVL.testintervalsecs := GVL.overall_cycle_time - REAL_TO_INT(chargeTIME + TIME_TO_REAL (extendedElapsed) + GVL.holdTIMEsec);
ELSE
	GVL.testintervalsecs := GVL.overall_cycle_time - REAL_TO_INT(GVL.chargeTIMEmanual + GVL.holdTIMEsec);
END_IF

//added sparkgap charger OFF when DUMP Relay is close sept 21, 2022 GL
(*IF GVL.softdump = FALSE THEN // NC, 0 = contact close, 1 = contact open
	GVL.sparkCharger_SP_Enable := FALSE; // turn off sparkcharge setpoint
	GVL.sparkCharger_ON := FALSE; // turn off sparkcharger
END_IF;*)

// Main Process Flow
IF GVL.appRUN THEN

	CASE processSTEP OF
		
		0:	(* FIRST RUN SETUP + WAIT 15 SEC *)
			GVL.softdump := FALSE;
			GVL.chargeCOIL := FALSE;
			GVL.psuInhibit := TRUE;
			volt_TO_AO1_802L50kV(psuTargetinvolt:= GVL.targetPSUVOLT, psuMaxOutput:= GVL.psuMaxOutput, VpsuOut:= GVL.psuVCTRL);	(* PSU setpoint function. *)
			GVL.shotCOIL := FALSE;
			GVL.scopetrigger := FALSE;
			
			IF GVL.softdump = FALSE THEN 
				GVL.sparkCharger_ON := FALSE;
				GVL.sparkCharger_SP_Enable := FALSE;
			END_IF;
			
			GVL.charging_alarm := TRUE;
			// Check temps
			cap1_Temp := tempSAFE(TEMPcel:= GVL.TEMPcap1, thresholdTEMPcel:= GVL.cap1THRESHOLDcel);
			dump_Temp := tempSAFE(TEMPcel:= GVL.TEMPdump, thresholdTEMPcel:= GVL.softdumpTHRESHOLDcel);
			load_Temp := tempSAFE(TEMPcel:= GVL.TEMPload, thresholdTEMPcel:= GVL.loadTHRESHOLDcel);
			ambient_Temp := tempSAFE(TEMPcel:= GVL.TEMPambient, thresholdTEMPcel:= GVL.ambientTHRESHOLDcel);
		
			// Wait before startinZg (Safety)
			IF cap1_Temp AND dump_Temp AND load_Temp AND ambient_Temp THEN
				beforestartTON(IN:= TRUE, PT:= firstwaitTIME, Q=> startReady, ET=> elapsedbeforestartTIME);
			ELSE
				beforestartTON(IN:= FALSE, PT:= firstwaitTIME, Q=> startReady, ET=> elapsedbeforestartTIME);
				elapsedbeforestartTIME := T#0MS;
			END_IF;
			// Proceed to next step
			IF (startReady AND GVL.HOA)		// Automatic Operation
				XOR
				(GVL.HMIcharge AND startReady AND NOT GVL.HOA)		// Manual Operation
				THEN
				beforestartTON(IN:= FALSE, PT:= firstwaitTIME, Q=> startReady, ET=> elapsedbeforestartTIME);
				elapsedbeforestartTIME := T#0S;
				lasttimesec := 0;
				GVL.charging_alarm := FALSE;
				GVL.chrg_to_fire_trig := FALSE;
				GVL.selectREMOTE := TRUE;		// psuHV On once at start, charging controlled by inhibit
				IF GVL.control_current THEN
					processSTEP := 6;
				ELSE
					processSTEP := 1;
				END_IF
			END_IF
			
		1: 	(* CHARGE *)
			// Increments test number once; tracked with internalBOOLcharge
			IF NOT internalBOOLcharge THEN
				GVL.testNUM := GVL.testNUM + 1;
				internalBOOLcharge := TRUE;
			END_IF
			
			// If Labview charge time set to -1 then use automatic/ estimated full charge time to V setpoint. Value > 0 is a manual charge time.
			estfullchrgTIME := estimatedchargeTIME_802L(uFcapacitance:= GVL.circuitcapacitanceuF, Vrated:= GVL.psuVOLTrating, Vcharge:= GVL.targetPSUVOLT, Powerpk802L:= GVL.psuPOWERpeak);	// In seconds
			IF GVL.chargeTIMEmanual >= 0 THEN
				chargeTIME := GVL.chargeTIMEmanual;	// Manual charge time, seconds
				fullCHRG := FALSE;
			ELSE
				chargeTIME := estfullchrgTIME;		// Full charging relies on PSU EOC signal	
				fullCHRG := TRUE;
			END_IF	
			// Error handling for chargeTIME == 0
			IF chargeTIME = 0 THEN
				GVL.appRUN := FALSE;
			END_IF
			chargeTIMEdint := REAL_TO_DINT((chargeTIME)*1000); // To millisec
			chargeTIMEtime := DINT_TO_TIME(chargeTIMEdint);		// To TIME
			
			expectcapVOLT := instantexpectedcapVOLT_802L(	// Expected cap voltage at instant time
				timenow:= elapsedCharge, 
				capacitanceF:= (GVL.circuitcapacitanceuF*0.001),
				PSUratedVoltage:= GVL.psuVOLTrating,
				targetVoltage:= GVL.targetPSUVOLT,  
				previoustime:= lasttimesec, 
				Voltlast:= capvoltiter); 
			
			GVL.Vcap1 := AI5volt(AI5voltageraw:= GVL.rawVcap1, isGreaterthanlimit:= GVL.changeAI5 );		// Get cap VOLT. Voltage interpreted as abs value.
			GVL.expectedvoltage := REAL_TO_INT(expectcapVOLT);
			// Start charge.
			// Algorithm that compares real voltage to the expected charge curve +/-500V. Charge too fast or charge too slow raises fault
			IF GVL.Vcap1 <= (expectcapVOLT+chrgvoltTOLERANCE) AND GVL.Vcap1 >= (expectcapVOLT-chrgvoltTOLERANCE)
				AND NOT GVL.psuONOFF THEN	
				GVL.softdump := TRUE; // NC
				
				IF GVL.softdump_contact THEN 		// ! Waits for not soft dumping
					GVL.chargeCOIL := TRUE;	
					GVL.chrg_to_fire_trig := TRUE;
					IF GVL.chargeCOIL_contact THEN
						chargeTON(IN:= TRUE, PT:= chargeTIMEtime, Q=> inhibitVariable, ET=> elapsedCharge );		// False until ET
						GVL.psuInhibit := FALSE;	// Equates on sepearate line to reduce flickering.
					END_IF;
				END_IF;
			ELSIF GVL.Vcap1 > (expectcapVOLT+chrgvoltTOLERANCE) OR GVL.Vcap1 < (expectcapVOLT-chrgvoltTOLERANCE) THEN
				GVL.chargeFAULT := TRUE;		// Fault handled below
			END_IF;
			//SCR FB Fault
			IF NOT GVL.isnotSCRhvswitch THEN
				GVL.Vcap1 := AI5volt(AI5voltageraw:= GVL.rawVcap1, isGreaterthanlimit:= GVL.changeAI5 );
				IF GVL.Vcap1 >= 5000 THEN 
					IF NOT GVL.shotCOILrdy THEN		// Need SCR rdy before shot
						GVL.dischargeFAULT := TRUE;
					END_IF
				END_IF;
			END_IF;
			(* Proceed to HOLD logic + EOC not reached FAULTS (Manual charge time holds when time reached. Automatic (-1) uses waits for EOC signal to hold)
			NOTE: EOC is normally high. 
			If the TDK charger is replaced in the future, the Glassman PSU exit logic can be placed here. *)
			elapsedChargereal := TIME_TO_REAL(elapsedCharge)*0.001;	// From ms to sec
 
			EOCF_TRIG(CLK:= GVL.EOCstatus, Q=> EOCBool);
			IF EOCBool OR iterateEOC THEN
				iterateEOC := TRUE;
				elapsedEOC := T#0S;
				EOCTON(IN:= TRUE, PT:= EOCTIMEtime, Q=> EOCBool2, ET=> elapsedEOC);
			END_IF
			IF EOCBool2 THEN
				EOCTON(IN:= FALSE, PT:= EOCTIMEtime, Q=> EOCBool2, ET=> elapsedEOC);
				elapsedEOC := T#0S;
				iterateEOC := FALSE;
				IF NOT GVL.EOCstatus THEN
					EOCPassed := TRUE;
				ELSE
					EOCPassed := FALSE;
				END_IF
			END_IF

			IF elapsedChargereal >= chargeTIME THEN
				extendedChargeTimer(IN :=TRUE, PT:= extendedToleranceTIME,Q => extendedTimeReached, ET =>extendedElapsed);
			END_IF;
			
			// This was changed on my last day! Replace EOCPassed with GVL.EOC Mind if NL or NH
			IF ((elapsedChargereal >= (chargeTIME*lowlimtimeTOLERANCE) ) AND EOCPassed AND GVL.Vcap1 >=GVL.targetPSUVOLT-300 AND NOT extendedTimeReached AND fullCHRG) 	// Automatic Operation - Goto HOLD
				OR ((elapsedChargereal >= chargeTIME) AND NOT fullCHRG)
				OR (GVL.HMIhold AND NOT GVL.HOA)		// Manual Operation - Can exit charge at any time. Will exit upon full charge reached even in manual operation.
				THEN
				
				EOCPassed := FALSE;
				EOCBool := FALSE;
				EOCBool2 := FALSE;
				EOCTON(IN:= FALSE, PT:= EOCTIMEtime, Q=> EOCBool2, ET=> elapsedEOC);
				extendedChargeTimer(IN :=FALSE, PT:= extendedToleranceTIME,Q => extendedTimeReached, ET =>extendedElapsed);
				extendedElapsed := T#0MS;
				chargeTON(IN:= FALSE, PT:= chargeTIMEtime, Q=> inhibitVariable, ET=> elapsedCharge );
				elapsedCharge := T#0MS;
				lasttimesec := 0;
				capvoltiter := 0;
				IF GVL.voltage_held_by_PSU THEN
					processSTEP := 2;
				ELSE
					GVL.psuInhibit := TRUE;
					GVL.chargeCOIL := FALSE;
					processSTEP :=7;
				END_IF;
				VoltAtHOLD := GVL.Vcap1;
				expectedATHOLD:= expectcapVOLT;
				internalBOOLcharge := FALSE;
			ELSIF  extendedTimeReached AND fullCHRG THEN //added in the event that EOC does not occur and cap keeps charging 
				GVL.chargeFAULT := TRUE;
			END_IF;
			
			// Handle the charge fault 
			IF  GVL.chargeFAULT THEN
				chargeTON(IN:= FALSE, PT:= chargeTIMEtime, Q=> inhibitVariable, ET=> elapsedCharge );
				elapsedCharge := T#0MS;
				internalBOOLcharge := FALSE;
				lasttimesec := 0;
				capvoltiter := 0;
			END_IF
			// Added pre-fire protection.  IF sample 2 is less than 5% of sample 1, go to dump State. Nov 09, 2022
			//*****************************************************
			FOR i := 1 TO 2 BY 1 DO
				IF heartbeat.pulse_ms = TRUE THEN
					Vcap_sample[i] := GVL.Vcap1;
				END_IF;
			END_FOR;
				
			IF Vcap_sample[2] < (Vcap_sample[1] - (0.05 * Vcap_sample[1])) THEN // IF Vcap1 suddenly drop morethan 5% of of the previous sample, go to dump state.
				GVL.appRUN := FALSE;
				GVL.PreFire_Fault := TRUE;  
				fbGetSystemTIME(timeLoDW => fileTIME.dwLowDateTime, timeHiDW => fileTIME.dwHighDateTime);
				sTIME := SYSTEMTIME_TO_STRING (FILETIME_TO_SYSTEMTIME (fileTime)); 
				processSTEP :=  4;
			END_IF;
	
			//*********************************************************
		2:	(* HOLD BEFORE SHOT - Shot specified time. Cap voltage held by HVPS *)
			IF GVL.control_current THEN
				PRG_FB_CTRL_PWM_OUT();
			END_IF
			(* GVL.softdump := TRUE; // Here to describe current state
			GVL.shotCOIL := FALSE; *)
			holdTIMEtime := REAL_TO_TIME(GVL.holdTIMEsec*1000);	// Hold for HMI specified TIME (Converts s to ms for use by TIME)
			
			holdTON(IN:= TRUE, PT:= holdTIMEtime, Q=> shotready, ET=> elapsedhold);
			
			// Proceed to shot
			GVL.Vcap1 := AI5volt(AI5voltageraw:= GVL.rawVcap1, isGreaterthanlimit:= GVL.changeAI5 );		// Get cap VOLT
			IF (shotready AND GVL.HOA)		// Automatic Operation
				XOR
				(GVL.HMIshoot AND NOT GVL.HOA)		// Manual Operation
				THEN
				
				(*IF (GVL.Vcap1 < (VoltAtHOLD-holdvoltThreshold)) THEN		// Cap volt leak fault
					GVL.holdFAULT := TRUE;
				END_IF*)
				internalBOOLSDL := TRUE;
				GVL.psuInhibit := TRUE;		// Diode reverse protected
				GVL.chargeCOIL := FALSE;
			ELSIF  (GVL.HMIdump OR shotready) AND NOT GVL.HOA THEN
				processSTEP := 5;
				internalBOOLSDL := FALSE;
			END_IF;
			
			holdTON2(IN:= internalBOOLSDL, PT:= T#1S, Q=> shotready2, ET=> elapsedhold2);
			
			IF shotready2 AND NOT GVL.chargeCOIL_contact THEN
				internalBOOLSDL := FALSE;
				holdTON2(IN:= FALSE, PT:= T#1S, Q=> shotready2, ET=> elapsedhold2);
				shotready2 := FALSE;
				elapsedhold2 := T#0S;
				
				IF GVL.isnotSCRhvswitch = FALSE THEN
					IF GVL.shotCOILrdy = FALSE THEN		// Need SCR rdy before shot
						GVL.dischargeFAULT := TRUE;
					END_IF;
				END_IF;
					
				IF GVL.isnotSCRhvswitch = TRUE THEN  //not SCR so we use sparkgap //Added spark charger enable
					GVL.sparkCharger_ON := TRUE;
					GVL.sparkCharger_SP_enable := TRUE;
					sparkcharger_TON (IN:= TRUE, PT:= sparkcharger_TON_PT, Q=> sparkcharger_ready);
					IF sparkcharger_ready THEN
						holdTON(IN:= FALSE, PT:= holdTIMEtime, Q=> shotready, ET=> elapsedhold); //added rev2
						shotready := FALSE;
						elapsedhold := T#0MS;
						
						processSTEP := 3;
					END_IF;	
				ELSE
					holdTON(IN:= FALSE, PT:= holdTIMEtime, Q=> shotready, ET=> elapsedhold);
					shotready := FALSE;
					elapsedhold := T#0MS;
					processSTEP :=3;
				END_IF;
				
			END_IF;
			
			
		3:	(* SHOT - automatically proceeeds to wait after shot *)
			sparkcharger_TON (IN:= FALSE, PT:= sparkcharger_TON_PT, Q=> sparkcharger_ready);
			GVl.sparkCharger_SP_Enable := FALSE; //Added Spark charger turn off right before the shooting.
			GVl.sparkCharger_ON := FALSE;
			
			
			GVL.chargeCOIL := FALSE;
			
			hold_betweenCharge_nShot_TON (IN:= TRUE, PT:= hold_betweenCharge_nShot_PT);
			
			IF hold_betweenCharge_nShot_TON.Q = TRUE THEN
				GVL.shotCOIL := TRUE;
				GVL.scopetrigger := TRUE;
				GVL.chrg_to_fire_trig:= FALSE;
			END_IF
			
			shotTON(IN:= TRUE, PT:= shotrelayDURATION, Q=> shooted, ET=> elapsedshot);	// Continue shot for 250ms
			IF shooted THEN
				IF GVL.isnotSCRhvswitch = FALSE THEN
					IF GVL.shotCOILrdy THEN		// SCR rdy is high if didn't shoot
						GVL.dischargeFAULT := TRUE;
					END_IF
				END_IF;
				
				shotTON(IN:= FALSE, PT:= shotrelayDURATION, Q=> shooted, ET=> elapsedshot);
				hold_betweenCharge_nShot_TON (IN:= FALSE, PT:= hold_betweenCharge_nShot_PT); 
				shooted := FALSE;
				elapsedshot := T#0MS;
				GVL.shotCOIL := FALSE;
				
				IF GVL.chargeCOIL_contact = FALSE THEN
					sparkcharger_softdump_TON (IN:= TRUE, PT:= sparkcharger_softdump_PT);
				
					IF sparkcharger_softdump_TON.Q = TRUE THEN
						processstep :=4;
					END_IF;
				END_IF;
				
				processstep :=4;				
			END_IF;	
			
		4:	(* WAIT TEST INTERVAL *)
			GVL.softdump := FALSE;	// NC
			IF GVL.softdump_contact = FALSE THEN
				GVL.sparkCharger_SP_Enable := FALSE; // turn off sparkcharge setpoint
				GVL.sparkCharger_ON := FALSE; // turn off sparkcharger
			END_IF;
			//GVL.softdump := FALSE;	// NC  - was here but added a timer.
			
			// Number of tests reached -> STOP
			IF GVL.testNUM >= GVL.testNUMmax THEN
				processSTEP := 0;
				GVL.appRUN := FALSE;
				GVL.testNUMexceed := TRUE;
			END_IF
			
			// Wait for safe temperatures
			waitTIMEtime := REAL_TO_TIME(INT_TO_REAL(GVL.testintervalsecs)*1000);		// LabVIEW input (s to ms for TIME)
			sparkcharger_softdump_TON (IN:= FALSE, PT:= sparkcharger_softdump_PT);
			testwaitTON(IN:= TRUE, PT:= waitTIMEtime, Q=> holdtimerQ, ET=> elapsedwait);
			cap1_Temp := tempSAFE(TEMPcel:= GVL.TEMPcap1, thresholdTEMPcel:= GVL.cap1THRESHOLDcel);
			dump_Temp := tempSAFE(TEMPcel:= GVL.TEMPdump, thresholdTEMPcel:= GVL.softdumpTHRESHOLDcel);
			load_Temp := tempSAFE(TEMPcel:= GVL.TEMPload, thresholdTEMPcel:= GVL.loadTHRESHOLDcel);
			ambient_Temp := tempSAFE(TEMPcel:= GVL.TEMPambient, thresholdTEMPcel:= GVL.ambientTHRESHOLDcel);
			
			//Sound charging alarm 5 sec before charge
			IF (elapsedwait >= (waitTIMEtime- T#5S)) THEN
				GVL.charging_alarm := TRUE;
			END_IF
			// Proceed to charge upon time delay AND safe temperatures
			IF ( (holdtimerQ AND GVL.HOA)		// Automatic Operation
				XOR (GVL.HMIcharge AND NOT GVL.HOA) )		// Manual Operation
				AND cap1_Temp AND dump_Temp AND load_Temp AND ambient_Temp THEN
				testwaitTON(IN:= FALSE, PT:= waitTIMEtime, Q=> holdtimerQ, ET=> elapsedwait);
				holdtimerQ := FALSE;
				elapsedhold := T#0MS;
				GVL.scopetrigger := FALSE;
				GVL.charging_alarm := FALSE;
				
				IF GVL.control_current THEN
					processSTEP := 6;
				ELSE
					processSTEP := 1;
				END_IF
				
			END_IF;
			
		5:
				GVL.appRUN := FALSE;
				
		6: //Control Current
			IF NOT internalBOOLcharge THEN
				GVL.testNUM := GVL.testNUM + 1;
				internalBOOLcharge := TRUE;
			END_IF
			estfullchrgTIME := estimatedchargeTIME_802L(uFcapacitance:= GVL.circuitcapacitanceuF, Vrated:= GVL.psuVOLTrating, Vcharge:= GVL.targetPSUVOLT, Powerpk802L:= GVL.psuPOWERpeak);	// In seconds
						
			IF GVL.chargeTIMEmanual >= 0 THEN
				chargeTIME := GVL.chargeTIMEmanual;	// Manual charge time, seconds
				fullCHRG := FALSE;
			ELSE
				chargeTIME := estfullchrgTIME;		// Full charging relies on PSU EOC signal	
				fullCHRG := TRUE;
			END_IF	
			// Error handling for chargeTIME == 0
			IF chargeTIME = 0 THEN
				GVL.appRUN := FALSE;
			END_IF
			chargeTIMEdint := REAL_TO_DINT((chargeTIME)*1000); // To millisec
			chargeTIMEtime := DINT_TO_TIME(chargeTIMEdint);		// To TIME
			
			expectcapVOLT := instantexpectedcapVOLT_802L(	// Expected cap voltage at instant time
				timenow:= elapsedCharge, 
				capacitanceF:= (GVL.circuitcapacitanceuF*0.001),
				PSUratedVoltage:= GVL.psuVOLTrating,
				targetVoltage:= GVL.targetPSUVOLT,  
				previoustime:= lasttimesec, 
				Voltlast:= capvoltiter); 
			
			GVL.Vcap1 := AI5volt(AI5voltageraw:= GVL.rawVcap1, isGreaterthanlimit:= GVL.changeAI5 );		// Get cap VOLT. Voltage interpreted as abs value.
			GVL.expectedvoltage := REAL_TO_INT(expectcapVOLT);
			
			IF (GVL.Vcap1 >= (GVL.expectedvoltage - 2000)) THEN
				GVL.softdump := TRUE;
				IF GVL.softdump_contact THEN 		// ! Waits for not soft dumping
					GVL.chargeCOIL := TRUE;
					GVL.chrg_to_fire_trig := TRUE;
					IF GVL.chargeCOIL_contact THEN
							chargeTON(IN:= TRUE, PT:= chargeTIMEtime, Q=> inhibitVariable, ET=> elapsedCharge );		// False until ET
							GVL.psuInhibit := FALSE;	// Equates on sepearate line to reduce flickering.
							PRG_FB_CTRL_PWM_OUT();
					END_IF;
				END_IF;
			ELSE
				GVL.chargeFAULT := TRUE;
			END_IF;
			//SCR FB Fault
			IF NOT GVL.isnotSCRhvswitch THEN
				GVL.Vcap1 := AI5volt(AI5voltageraw:= GVL.rawVcap1, isGreaterthanlimit:= GVL.changeAI5 );
				IF GVL.Vcap1 >= 5000 THEN 
					IF NOT GVL.shotCOILrdy THEN		// Need SCR rdy before shot
						GVL.dischargeFAULT := TRUE;
					END_IF
				END_IF;
			END_IF;
			elapsedChargereal := TIME_TO_REAL(elapsedCharge)*0.001;
			IF elapsedChargereal >= GVL.chargeTIMEmanual OR (GVL.HMIhold AND NOT GVL.HOA) THEN
				chargeTON(IN:= FALSE, PT:= chargeTIMEtime, Q=> inhibitVariable, ET=> elapsedCharge );
				elapsedCharge := T#0MS;
				IF GVL.voltage_held_by_PSU THEN
					processSTEP := 2;
				ELSE
					GVL.psuInhibit := TRUE;
					GVL.chargeCOIL := FALSE;
					processSTEP :=7;
				END_IF;
				VoltAtHOLD := GVL.Vcap1;
				expectedATHOLD:= expectcapVOLT;
				internalBOOLcharge := FALSE;
			END_IF
			// Handle the charge fault 
			IF  GVL.chargeFAULT THEN
				chargeTON(IN:= FALSE, PT:= chargeTIMEtime, Q=> inhibitVariable, ET=> elapsedCharge );
				elapsedCharge := T#0MS;
				internalBOOLcharge := FALSE;
			END_IF
			
			// Added pre-fire protection.  IF sample 2 is less than 5% of sample 1, go to dump State. Nov 09, 2022
			//*****************************************************
			
			FOR i := 1 TO 2 BY 1 DO
				IF heartbeat.pulse_ms = TRUE THEN
					Vcap_sample[i] := GVL.Vcap1;
				END_IF;
			END_FOR;
				
			IF Vcap_sample[2] < (Vcap_sample[1] - (0.05 * Vcap_sample[1])) THEN // IF Vcap1 suddenly drop morethan 5% of of the previous sample, go to dump state.
				
				GVL.appRUN := FALSE;
				GVL.PreFire_Fault := TRUE;  
				fbGetSystemTIME(timeLoDW => fileTIME.dwLowDateTime, timeHiDW => fileTIME.dwHighDateTime);
				sTIME := SYSTEMTIME_TO_STRING (FILETIME_TO_SYSTEMTIME (fileTime)); 
				processSTEP :=  4;  
			END_IF;
		
			//*********************************************************
			
		7: (* HOLD BEFORE SHOT - Shot specified time. Cap open circuited and not voltage held by HVPS *)
			GVL.psuInhibit := TRUE;		// Diode reverse protected
			GVL.chargeCOIL := FALSE;
			(* GVL.softdump := TRUE; // Here to describe current state
			GVL.shotCOIL := FALSE; *)
			holdTIMEtime := REAL_TO_TIME(GVL.holdTIMEsec*1000);	// Hold for HMI specified TIME (Converts s to ms for use by TIME)
			holdTON(IN:= TRUE, PT:= holdTIMEtime, Q=> shotready, ET=> elapsedhold);
			
			// Proceed to shot
			GVL.Vcap1 := AI5volt(AI5voltageraw:= GVL.rawVcap1, isGreaterthanlimit:= GVL.changeAI5 );	// Get cap VOLT
			IF (shotready AND GVL.HOA)		// Automatic Operation
				XOR
				(GVL.HMIshoot AND NOT GVL.HOA)		// Manual Operation
				THEN
				
				IF GVL.Vcap1 < (VoltAtHOLD-holdvoltThreshold) THEN		// Cap volt leak fault
					GVL.holdFAULT := TRUE;
				END_IF
				
				IF NOT GVL.isnotSCRhvswitch THEN
					IF NOT GVL.shotCOILrdy THEN		// Need SCR rdy before shot
						GVL.dischargeFAULT := TRUE;
					END_IF
				END_IF;
				
				holdTON(IN:= FALSE, PT:= holdTIMEtime, Q=> shotready, ET=> elapsedhold);
				shotready := FALSE;
				elapsedhold := T#0MS;
				processstep := 3;
			ELSIF	(GVL.HMIdump OR shotready) AND NOT GVL.HOA THEN
				processSTEP := 5;
			END_IF;
			
		99:
			// HMI Invalid HMI Entries should be handled within LabVIEW. Case 99 not used - For expansion of error handling
			processSTEP := 0;
			GVL.appRUN := FALSE;
			GVL.softdump := FALSE;
			GVL.psuONOFF := FALSE; 
			GVL.psuInhibit := TRUE;
			GVL.shotCOIL := FALSE;
			volt_TO_AO1_802L50kV(psuTargetinvolt:= 0, psuMaxOutput:= GVL.psuMaxOutput, VpsuOut:= GVL.psuVCTRL);
			GVL.ctrlsysFAULT := TRUE;
			
	END_CASE;
	
	IF i > 2 THEN
		i := 1;
	END_IF;
END_IF;

END_PROGRAM

// ---- POUs/Functions/AnalogOut-ScaleOffset/volt_TO_AO1_802L50kV.TcPOU
FUNCTION volt_TO_AO1_802L50kV : INT
VAR_INPUT
	psuTargetinvolt : DINT;
	psuMaxOutput : UINT;
END_VAR
VAR_IN_OUT
	VpsuOut : INT;
END_VAR
VAR
	x_min 					: REAL;
	psuTargetinvolt_REAL 	: REAL;
	psuMaxOutput_REAL 		: REAL;
	VpsuOUT_REAL 			: REAL;
END_VAR

(* Description:
Converts voltage to respective AO1 0-32767 sig
Specific to the negative TDK 802L 12kV, 12kV is 802L max out. 32767 is 10V PLC out. *)

(* Min setpoint ~0.5kV due to 17-0066E 
!! Must be recalibrated for any other PSU!! *)

// Build for 17-0066E
psuTargetinvolt := ABS(psuTargetinvolt);
IF psuTargetinvolt > psuMaxOutput THEN	
	psuTargetinvolt := psuMaxOutput;
END_IF

//VpsuOUT := REAL_TO_INT( (DINT_TO_REAL(psuTargetinvolt) + 20.0 ) / 0.38745387453874538744);
// For +50kV PSU: VpsuOUT := REAL_TO_INT( (DINT_TO_REAL(psuTargetinvolt)-99.009) / 1.5841584158415841584);
//VpsuOUT := REAL_TO_INT( (DINT_TO_REAL(psuTargetinvolt)*2.730583333333333333333333));
psuTargetinvolt_REAL := DINT_TO_REAL (psuTargetinvolt);
psuMaxOutput_REAL := UINT_TO_REAL (psuMaxOutput);

VpsuOUT_REAL := 32767 * (psuTargetinvolt_REAL - x_min) / (psuMaxOutput_REAL - x_min);

VpsuOUT := REAL_TO_INT (VpsuOUT_REAL);

//set the limit for AQ over range  - This should never happen.
IF VpsuOUT > 32767 THEN
	VpsuOUT := 32767;
END_IF;

IF VpsuOUT < 0 THEN		// Block negative voltage out
	VpsuOUT := 0;
END_IF;

END_FUNCTION

// ---- POUs/Functions/estimatedchargeTIME_802L.TcPOU
FUNCTION estimatedchargeTIME_802L : REAL
VAR_INPUT
	uFcapacitance : REAL;		// uF
	Vrated : DINT;				// Volts
	Vcharge : DINT;				// Volts
	Powerpk802L : REAL := 9000;	// J/s
END_VAR
VAR
END_VAR

(* Returns estimated charge time in seconds.
Using TDK 802L constant current stage 1 + power stage 2. *)

// LabVIEW set Ppeak802L to >= 1 to avoid error/ division by 0. Implemented for safety.
IF Powerpk802L = 0 THEN
	estimatedchargeTIME_802L := 0;
ELSE
	estimatedchargeTIME_802L := 0.5*uFcapacitance*0.000001*DINT_TO_REAL(Vrated*Vcharge)/Powerpk802L;
END_IF

END_FUNCTION

// ---- POUs/Functions/instantexpectedcapVOLT_802L.TcPOU
FUNCTION instantexpectedcapVOLT_802L : REAL
VAR_INPUT
	timenow : TIME;
	capacitanceF : REAL;
	PSUratedVoltage : DINT;
	targetVoltage : DINT;
END_VAR
VAR_IN_OUT
	previoustime : REAL;
	Voltlast : REAL;
END_VAR
VAR
	timenowsec : REAL;
	Powerpeak802L : REAL := 9000;
	timestepsec : REAL;
	Ipeak : REAL;
	I : REAL;
END_VAR

(* Function specific to TDK 802L. Must be modified for other models. 
Assumed to using the constant charging and constant power scheme. *)

timenowsec := TIME_TO_REAL(timenow)*0.001;	// From ms to sec
IF PSUratedVoltage = 0 THEN
	instantexpectedcapVOLT_802L := 0;
ELSE
	Ipeak := 2.0*Powerpeak802L/DINT_TO_REAL(PSUratedVoltage);
	timestepsec := timenowsec-previoustime;
	// Return last known voltage if timestep is 0
	IF targetVoltage <= 6000 THEN
		I := Ipeak;
	ELSE
		I := Ipeak*(0.5+(DINT_TO_REAL(PSUratedVoltage)-Voltlast)/DINT_TO_REAL(PSUratedVoltage));
	END_IF
	IF timestepsec >= 0 THEN
		previoustime := previoustime+timestepsec;
		Voltlast := timestepsec/capacitanceF*I+Voltlast;
	END_IF
	IF Voltlast >= DINT_TO_REAL(targetVoltage) THEN
		instantexpectedcapVOLT_802L := DINT_TO_REAL(targetVoltage);
	ELSE
		instantexpectedcapVOLT_802L := Voltlast;
	END_IF;
END_IF

END_FUNCTION

// ---- POUs/PRG_FB_CTRL_PWM_OUT.TcPOU
PROGRAM PRG_FB_CTRL_PWM_OUT
VAR
	fPwmInput					: LREAL := 50;
	bPwmOutBitPos				: BOOL;
	bPwmOutBitNeg				: BOOL;

	fbCTRL_PWM_OUT				: FB_CTRL_PWM_OUT;
	stCTRL_PWM_OUT_PARAMS		: ST_CTRL_PWM_OUT_PARAMS;

	eMode						: E_CTRL_MODE;
	eErrorId					: E_CTRL_ERRORCODES;
	bError						: BOOL;

	bInit						: BOOL	:= TRUE;
	fDelta						: LREAL	:= 0.05;
END_VAR

IF bInit THEN
	(* init parameter struct *)
	stCTRL_PWM_OUT_PARAMS.tTaskCycleTime	:= T#10MS;
	stCTRL_PWM_OUT_PARAMS.tPWMPeriod		:= T#1S;

	(* set the mode to ACTIVE --> normal operation *)
	eMode := eCTRL_MODE_ACTIVE;

	(* reset the init flag *)
	bInit := FALSE;
END_IF
fPwmInput := GVL.duty_cycle;
fbCTRL_PWM_OUT(	fPwmInput			:= fPwmInput,
				eMode				:= eMode,
				stParams			:= stCTRL_PWM_OUT_PARAMS,
				bPwmOutBitPos		=> bPwmOutBitPos,
				bPwmOutBitNeg		=> bPwmOutBitNeg,
				bError				=> bError,
				eErrorId			=> eErrorId);


(* copy var to scope var *)
GVL.psuInhibit := NOT bPWMOutBitPos;
//bPWMNegOutToScope := bPWMOutBitNeg;

END_PROGRAM

// ---- POUs/handlesensorlimitFAULTS.TcPOU
PROGRAM handlesensorlimitFAULTS
VAR
END_VAR

(* Handles instrumentation faults.
Program looks at the lower and upper limit bits on each sensor channel.
The temperature sensors using the 17-0284 PCBs give an approx .8-10V signal. Anything below 4mA or .8V means that the PCB/ sensor has failed  

4mA PWM signal ~= .8V. The EL3XXX is set to 1000 lower limit
*)
IF (GVL.PLC_AI1_LIM1.2		// BIt_0 is the lower limit fault.
OR GVL.PLC_AI2_LIM1.2
OR GVL.PLC_AI3_LIM1.2
OR GVL.PLC_AI4_LIM1.2 
) THEN
	GVL.InstrumentationFault := TRUE;
END_IF

END_PROGRAM

// ---- POUs/handlesoftEXCEPTION.TcPOU
PROGRAM handlesoftEXCEPTION
VAR
	zero : LREAL := 0.000000001;	// Account for floating point representation
END_VAR

(* Handle firmware/HMI exceptions by stopping GVL.appRUN *)

// Handle HMI invalid ranges
IF GVL.chargeTIMEmanual < -1 OR GVL.circuitcapacitanceuF <= zero OR GVL.targetPSUVOLT <= zero OR GVL.psuVOLTrating <= zero OR GVL.psuPOWERpeak <= zero OR GVL.chargeTIMEmanual >60 THEN
	GVL.ctrlsysFAULT := TRUE;
	GVL.softexceptionFAULT:= TRUE;
END_IF

END_PROGRAM

// ---- POUs/HMI.TcPOU
PROGRAM HMI
VAR
END_VAR

IF GVL.appRUN = FALSE AND GVL.noFaultDetected = TRUE THEN 
	GVL.chargeCOIL := HMI_DB.ActivateChargePB;
	GVL.softdump 	:= HMI_DB.ActivateDumpPB;
	END_IF
	
//FAULTS - Underdevelopment

HMI_DB.Fault.0 := GVL.sparkdetect;
HMI_DB.Fault.1 := GVL.FireDetected;

//HMI_DB.Fault.2 := 
//HMI_DB.Fault.3 := 

//TRIPS



//PERMISSIVES


//HMI bit mapping
HMI_DB.Charging := GVL.chargeCOIL_contact;
HMI_DB.Dumping := NOT GVL.softdump_contact;

(*IF GVL.softdump_contact = FALSE THEN  //softdump_contact is normally closed.  When closed, dumping coil is open.
	HMI_DB.Dumping := TRUE;
ELSE
	HMI_DB.Dumping := FALSE;
END_IF;*)

END_PROGRAM

// ---- POUs/Functions/HV_Monitor.TcPOU
PROGRAM HV_Monitor
VAR
	scaled_voltage :INT;
	avg_raw : INT;
	sum_raw : REAL;
	prev_raw : INT;
	i : INT:=0;
END_VAR

//scaled_voltage := REAL_TO_INT(1.6433*raw-12270);
//scaled_voltage := REAL_TO_INT(1.6577*raw-12721);
(*IF (GVL.raw_HV_monitor<=7180 AND GVL.raw_HV_monitor>=7040) THEN
	sum_raw:=0;
	FOR i := 1 TO 20{BY 1)} DO
		sum_raw:= sum_raw+GVL.raw_HV_monitor ;
	END_FOR
	avg_raw:=REAL_TO_INT((sum_raw)/20);
	IF (avg_raw <=7151 AND avg_raw>=7070) THEN
		scaled_voltage:=0; 
	ELSIF (avg_raw <=7116 AND avg_raw>=7052) THEN
		scaled_voltage:=-35;
	ELSIF (avg_raw <=7178 AND avg_raw>=7080) THEN
		scaled_voltage:=35;
	END_IF
ELSE
	scaled_voltage := REAL_TO_INT(0.4748150*GVL.raw_HV_monitor-3558.738574);
END_IF*)
scaled_voltage := REAL_TO_INT(0.4748150*GVL.raw_HV_monitor-3558.738574);

END_PROGRAM

// ---- POUs/VoltMonitor.TcPOU
PROGRAM VoltMonitor
VAR
	i : USINT := 0;
	k : USINT := 0;
	counter : USINT := 0;
	b : ARRAY[0..3] OF BOOL;
	b1 : BOOL;
	b2 : BOOL;
	b3 : BOOL;
	pause : BOOL;
	

	
END_VAR


(*IF Heartbeat.pulse_ms = TRUE AND pause = FALSE THEN
	i := i + 1;
	counter := 16-i;
	IF counter >= 16 THEN 
		counter := 0;
	END_IF
	VoltMonitor_DB.Channel := counter ;
	VoltMonitor_DB.VoltageReading_raw[counter] := GVL.raw_VoltageMonitor;
END_IF*)

b[0] := 0; //VoltMonitor_DB.Channel.0;
b[1] := 0; //VoltMonitor_DB.Channel.1;
b[2] := 0; //VoltMonitor_DB.Channel.2;
b[3] := 0; //VoltMonitor_DB.Channel.3;
//VoltMonitor_DB.VoltageReading_raw[0] := GVL.raw_VoltageMonitor;


//VoltMonitor_DB.CapRaw_Str :=  MID (UINT_TO_STRING (GVL.B170357_CapRaw), 10, 5);



//VoltMonitor_DB.VoltageReading_raw[0] := VoltMonitor_DB.CapRaw; //STRING_TO_INT (VoltMonitor_DB.CapRaw_Str);
FOR k := 0 TO 24 BY 1 DO
	
	IF GVL.B170357_CapRaw[k] <> 0 THEN
		VoltMonitor_DB.VoltageReading_raw[k].0 := VoltMonitor_DB.CapRaw[k].2;
		VoltMonitor_DB.VoltageReading_raw[k].1 := VoltMonitor_DB.CapRaw[k].3;
		VoltMonitor_DB.VoltageReading_raw[k].2 := VoltMonitor_DB.CapRaw[k].4;
		VoltMonitor_DB.VoltageReading_raw[k].3 := VoltMonitor_DB.CapRaw[k].5;
	
		VoltMonitor_DB.VoltageReading_raw[k].4 := VoltMonitor_DB.CapRaw[k].6;
		VoltMonitor_DB.VoltageReading_raw[k].5 := VoltMonitor_DB.CapRaw[k].7;
		VoltMonitor_DB.VoltageReading_raw[k].6 := VoltMonitor_DB.CapRaw[k].8;
		VoltMonitor_DB.VoltageReading_raw[k].7 := VoltMonitor_DB.CapRaw[k].9;
	
		VoltMonitor_DB.VoltageReading_raw[k].8 := VoltMonitor_DB.CapRaw[k].10;
		VoltMonitor_DB.VoltageReading_raw[k].9 := VoltMonitor_DB.CapRaw[k].11;
	
		VoltMonitor_DB.VoltageReading_raw[k].10 := 0;//VoltMonitor_DB.CapRaw.14;
		VoltMonitor_DB.VoltageReading_raw[k].11 := 0;//VoltMonitor_DB.CapRaw.15;
		VoltMonitor_DB.VoltageReading_raw[k].12 := 0;//VoltMonitor_DB.CapRaw.12;
		VoltMonitor_DB.VoltageReading_raw[k].13 := 0;//VoltMonitor_DB.CapRaw.13;
		VoltMonitor_DB.VoltageReading_raw[k].14 := 0; //VoltMonitor_DB.CapRaw.14;
	
		VoltMonitor_DB.VoltageReading_raw[k].15 := 0;//VoltMonitor_DB.CapRaw.4;
		VoltMonitor_DB.CapRaw_DummySnap[k] := GVL.B170357_CapRaw[k];//VoltMonitor_DB.VoltageReading_raw[0];
		ELSE
			//VoltMonitor_DB.VoltageReading_raw[k] := 0;
			//VoltMonitor_DB.CapRaw_DummySnap[k] := 0;
	END_IF
	
END_FOR

//missedCTU.PV := 10000;
//missedCTU.RESET := FALSE;

IF GVL.B170357_CapRaw[1] <> GVL.B170357_CapRaw[11] OR 
	GVL.B170357_CapRaw[2] <> GVL.B170357_CapRaw[12] OR 
	GVL.B170357_CapRaw[2] <> GVL.B170357_CapRaw[13] OR 
	GVL.B170357_CapRaw[3] <> GVL.B170357_CapRaw[14] OR 
	GVL.B170357_CapRaw[3] <> GVL.B170357_CapRaw[15] OR 
	GVL.B170357_CapRaw[1] <> GVL.B170357_CapRaw[16] //OR 
	(*GVL.B170357_CapRaw[1] <> GVL.B170357_CapRaw[13]*) THEN
	VoltMonitor_DB.missedCTU.CU := TRUE;
	//VoltMonitor_DB.ONS (CLK := TRUE);
	ELSE
		VoltMonitor_DB.missedCTU.CU := FALSE;
		//VoltMonitor_DB.ONS.CLK := FALSE; 
END_IF

VoltMonitor_DB.missingCNT_REAL := WORD_TO_REAL(VoltMonitor_DB.missingCNT);
CounterUP();

//missingCNT := missedCTU.CV;

IF pause = TRUE THEN
	VoltMonitor_DB.VoltageReading_raw[0] := 0;
END_IF;

IF i > 16 THEN 
	i := 0;
END_IF

IF k > 24 THEN 
	k := 0;
END_IF

END_PROGRAM

// ---- POUs/CounterUP.TcPOU
PROGRAM CounterUP
VAR

END_VAR

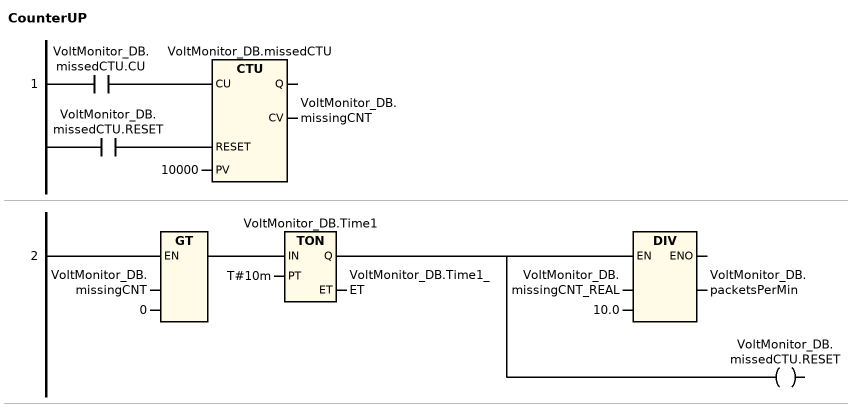
// NETWORK 1
VoltMonitor_DB.missedCTU(
    CU := VoltMonitor_DB.missedCTU.CU,
    RESET := VoltMonitor_DB.missedCTU.RESET,
    PV := 10000,
    CV => VoltMonitor_DB.missingCNT); // CTU

// NETWORK 2
VoltMonitor_DB.Time1(IN := VoltMonitor_DB.missingCNT > 0, PT := T#10m, ET => VoltMonitor_DB.Time1_ET); // TON
IF VoltMonitor_DB.Time1.Q THEN VoltMonitor_DB.packetsPerMin := VoltMonitor_DB.missingCNT_REAL / 10.0; END_IF
VoltMonitor_DB.missedCTU.RESET := VoltMonitor_DB.Time1.Q;

END_PROGRAM

// ---- POUs/ADC_5V.TcPOU
FUNCTION ADC_5V : REAL
VAR_INPUT
	normal_input : REAL;
	x_max : REAL := 4.5;
	x_min : REAL := 0.5;
END_VAR
VAR
	voltage_reading : REAL;
END_VAR

// 0.5 - 4.5V AI INPUT  | normal_input 0 - 100%
voltage_reading := 4.5 * normal_input;
ADC_5V := (voltage_reading - x_min) / (x_max - x_min);

END_FUNCTION

// ---- POUs/Functions/Norm_x_UINT.TcPOU
FUNCTION Norm_x_UINT : REAL
VAR_INPUT
	raw_input : REAL;
	x_max : UINT := 32767;  //for AI, use 32767, for AQ, use 12,000 or 50,000 V.
	x_min : UINT := 0;
END_VAR
VAR
END_VAR

// 0 - 12kV or 50kV input 
Norm_x_UINT := (raw_input - x_min) / (x_max - x_min);

END_FUNCTION
